		///////////АО КЦ от ШКС-04М////////////////////////////////////////////////////////////////////////
		//{name:АО КЦ от ШКС-04М}
		AOKC_SHKC:singleSignal(table:=ADR(imTable)):=(signal:=di.di_20.bits[0]);
		//{name:Обрыв сигнала "АО КЦ от ШКС-04М"}
		AOKC_SHKC_NS:Reability(table:=ADR(imTable)):=(di1:=di.di_9.bits[3], when:=FALSE);
		//{name:Наличие ЦК "АО КЦ от ШКС-04М"}
		AOKC_SHKC_CK:Reability(table:=ADR(imTable)):=(di1:=di.di_9.bits[3], when:=TRUE);
		
		///////////НО ГПА от кнопки на ШУ////////////////////////////////////////////////////////////////////////
		//{name:НО ГПА от кнопки на ШУ}
		NO_fromSHU:singleSignal(table:=ADR(imTable)):=(signal:=di.di_21.bits[1]);
		//{name:Обрыв сигнала "НО ГПА от кнопки на ШУ"}
		NO_fromSHU_NS:Reability(table:=ADR(imTable)):=(di1:=di.di_9.bits[4], when:=FALSE);
		//{name:Наличие ЦК  "НО ГПА от кнопки на ШУ"}
		NO_fromSHU_CK:Reability(table:=ADR(imTable)):=(di1:=di.di_9.bits[4], when:=TRUE);
		
		///////////АО ГПА от кнопки на ШУ////////////////////////////////////////////////////////////////////////
		//{name:АО ГПА от кнопки на ШУ}
		AO_fromSHU:singleSignal(table:=ADR(imTable)):=(signal:=di.di_21.bits[2]);
		//{name:Обрыв сигнала "АО ГПА от кнопки на ШУ"}
		AO_fromSHU_NS:Reability(table:=ADR(imTable)):=(di1:=di.di_9.bits[5], when:=FALSE);
		//{name:Наличие ЦК  "АО ГПА от кнопки на ШУ"}
		AO_fromSHU_CK:Reability(table:=ADR(imTable)):=(di1:=di.di_9.bits[5], when:=TRUE);
		
		///////////АО ЭГПА от ПРУ////////////////////////////////////////////////////////////////////////
		//{name:АО ЭГПА от ПРУ}
		AO_PRU:singleSignal(table:=ADR(imTable)):=(signal:=di.di_21.bits[3]);
		//{name:Обрыв сигнала "АО ЭГПА от ПРУ"}
		AO_PRU_NS:Reability(table:=ADR(imTable)):=(di1:=di.di_9.bits[6], when:=FALSE);
		//{name:Наличие ЦК "АО ЭГПА от ПРУ"}
		AO_PRU_CK:Reability(table:=ADR(imTable)):=(di1:=di.di_9.bits[6], when:=TRUE);
		
		///////////НКУ ввод 1 включен////////////////////////////////////////////////////////////////////////
		//{name:НКУ ввод 1 включен}
		NKU_1_On:singleSignal(table:=ADR(imTable)):=(signal:=di.di_10.bits[4]);
		//{name:Обрыв сигнала "НКУ ввод 1 включен"}
		NKU_1_On_NS:Reability(table:=ADR(imTable)):=(di1:=di.di_10.bits[4], when:=FALSE);
		//{name:Наличие ЦК  "НКУ ввод 1 включен"}
		NKU_1_On_CK:Reability(table:=ADR(imTable)):=(di1:=di.di_10.bits[4], when:=TRUE);
		
		///////////НКУ ввод 2 включен////////////////////////////////////////////////////////////////////////
		//{name:НКУ ввод 2 включен}
		NKU_2_On:singleSignal(table:=ADR(imTable)):=(signal:=di.di_10.bits[5]);
		//{name:Обрыв сигнала "НКУ ввод 2 включен"}
		NKU_2_On_NS:Reability(table:=ADR(imTable)):=(di1:=di.di_10.bits[5], when:=FALSE);
		//{name:Наличие ЦК  "НКУ ввод 2 включен"}
		NKU_2_On_CK:Reability(table:=ADR(imTable)):=(di1:=di.di_10.bits[5], when:=TRUE);
		///////////Неисправность цепей контроля ИМ////////////////////////////////////////////////////////////////////////
		MVvkl_Obryv_CK_NS:Reability(table:=ADR(imTable)):=(di1:=di.di_7.bits[0], when:=FALSE);
		MVvykl_Obryv_CK_NS:Reability(table:=ADR(imTable)):=(di1:=di.di_7.bits[1], when:=FALSE);
		MVControl_Work_Obryv_CK_NS:Reability(table:=ADR(imTable)):=(di1:=di.di_7.bits[2], when:=FALSE);
		PNS_vkl_CK_NS:Reability(table:=ADR(imTable)):=(di1:=di.di_5.bits[0], when:=FALSE);
		NU1_vkl_CK_NS:Reability(table:=ADR(imTable)):=(di1:=di.di_5.bits[1], when:=FALSE);
		NU2_vkl_CK_NS:Reability(table:=ADR(imTable)):=(di1:=di.di_5.bits[2], when:=FALSE);
		AVOM1_vkl_CK_NS:Reability(table:=ADR(imTable)):=(di1:=di.di_5.bits[3], when:=FALSE);
		AVOM2_vkl_CK_NS:Reability(table:=ADR(imTable)):=(di1:=di.di_5.bits[4], when:=FALSE);
		AVOM3_vkl_CK_NS:Reability(table:=ADR(imTable)):=(di1:=di.di_5.bits[5], when:=FALSE);
		AVOM4_vkl_CK_NS:Reability(table:=ADR(imTable)):=(di1:=di.di_5.bits[6], when:=FALSE);
		TEN_MB_vkl_CK_NS:Reability(table:=ADR(imTable)):=(di1:=di.di_10.bits[0], when:=FALSE);
		TEN_Kollectora_vkl_CK_NS:Reability(table:=ADR(imTable)):=(di1:=di.di_10.bits[1], when:=FALSE);
		Kalorifer_AVOM_vkl_CK_NS:Reability(table:=ADR(imTable)):=(di1:=di.di_10.bits[2], when:=FALSE);
		CMN_vkl_CK_NS:Reability(table:=ADR(imTable)):=(di1:=di.di_10.bits[3], when:=FALSE);
		///////////Наличие цепей контроля ИМ////////////////////////////////////////////////////////////////////////
		MVvkl_NAlichie_CK:Reability(table:=ADR(imTable)):=(di1:=di.di_7.bits[0], when:=TRUE);
		MVvykl_NAlichie_CK:Reability(table:=ADR(imTable)):=(di1:=di.di_7.bits[1], when:=TRUE);
		MVControl_Work_NAlichie_CK:Reability(table:=ADR(imTable)):=(di1:=di.di_7.bits[2], when:=TRUE);
		PNS_vkl_NAlichie_CK:Reability(table:=ADR(imTable)):=(di1:=di.di_5.bits[0], when:=TRUE);
		NU1_vkl_NAlichie_CK:Reability(table:=ADR(imTable)):=(di1:=di.di_5.bits[1], when:=TRUE);
		NU2_vkl_NAlichie_CK:Reability(table:=ADR(imTable)):=(di1:=di.di_5.bits[2], when:=TRUE);
		AVOM1_vkl_NAlichie_CK:Reability(table:=ADR(imTable)):=(di1:=di.di_5.bits[3], when:=TRUE);
		AVOM2_vkl_NAlichie_CK:Reability(table:=ADR(imTable)):=(di1:=di.di_5.bits[4], when:=TRUE);
		AVOM3_vkl_NAlichie_CK:Reability(table:=ADR(imTable)):=(di1:=di.di_5.bits[5], when:=TRUE);
		AVOM4_vkl_NAlichie_CK:Reability(table:=ADR(imTable)):=(di1:=di.di_5.bits[6], when:=TRUE);
		TEN_MB_vkl_NAlichie_CK:Reability(table:=ADR(imTable)):=(di1:=di.di_10.bits[0], when:=TRUE);
		TEN_Kollectora_vkl_NAlichie_CK:Reability(table:=ADR(imTable)):=(di1:=di.di_10.bits[1], when:=TRUE);
		Kalorifer_AVOM_vkl_NAlichie_CK:Reability(table:=ADR(imTable)):=(di1:=di.di_10.bits[2], when:=TRUE);
		CMN_vkl_NAlichie_CK:Reability(table:=ADR(imTable)):=(di1:=di.di_10.bits[3], when:=TRUE);
		///////////Наличие питания////////////////////////////////////////////////////////////////////////
		//{name:Наличие БП1}
		NalichieBP1:singleSignal(table:=ADR(imTable)):=(signal:=di.di_11.bits[0]);
		//{name:Наличие БП2}
		NalichieBP2:singleSignal(table:=ADR(imTable)):=(signal:=di.di_11.bits[1]);
		//{name:Наличие БП3}
		NalichieBP3:singleSignal(table:=ADR(imTable)):=(signal:=di.di_11.bits[2]);
		//{name:Наличие БП4}
		NalichieBP4:singleSignal(table:=ADR(imTable)):=(signal:=di.di_11.bits[3]);
		//{name:Наличие БП5}
		NalichieBP5:singleSignal(table:=ADR(imTable)):=(signal:=di.di_11.bits[4]);
		//{name:Наличие БП6}
		NalichieBP6:singleSignal(table:=ADR(imTable)):=(signal:=di.di_11.bits[5]);
		//{name:Наличие БП7 и БП8}
		NalichieBP7_BP8:singleSignal(table:=ADR(imTable)):=(signal:=di.di_11.bits[6]);
		//{name:Наличие БП9 и БП10}
		NalichieBP9_BP10:singleSignal(table:=ADR(imTable)):=(signal:=di.di_11.bits[7]);
		//{name:Наличие Цепи управления МВ}
		Nalichie_CU_MV:singleSignal(table:=ADR(imTable)):=(signal:=di.di_12.bits[0]);
		//{name:Наличие напряжения  =220 в БРЭО}
		Nalichie220BEAO:singleSignal(table:=ADR(imTable)):=(signal:=di.di_12.bits[1]);
		//{name:Наличие напряжения на входе в ШУ ~220}
		NalichiePer220naVhode:singleSignal(table:=ADR(imTable)):=(signal:=di.di_12.bits[2]);
		//{name:Наличие напряжения на входе в ШУ =220}
		NalichiePost220naVhode:singleSignal(table:=ADR(imTable)):=(signal:=di.di_12.bits[3]);
		//{name:Наличие БП11}
		NalichieBP11:singleSignal(table:=ADR(imTable)):=(signal:=di.di_12.bits[4]);
		//{name:Наличие БП12}
		NalichieBP12:singleSignal(table:=ADR(imTable)):=(signal:=di.di_12.bits[5]);
		
		///////////Отсутствие питания////////////////////////////////////////////////////////////////////////
		//{name:Нет БП1}
		NalichieBP1_NS:singleSignal(table:=ADR(imTable)):=(signal:=di.di_11.bits[0].inverse);
		//{name:Нет БП2}
		NalichieBP2_NS:singleSignal(table:=ADR(imTable)):=(signal:=di.di_11.bits[1].inverse);
		//{name:Нет БП3}
		NalichieBP3_NS:singleSignal(table:=ADR(imTable)):=(signal:=di.di_11.bits[2].inverse);
		//{name:Нет БП4}
		NalichieBP4_NS:singleSignal(table:=ADR(imTable)):=(signal:=di.di_11.bits[3].inverse);
		//{name:Нет БП5}
		NalichieBP5_NS:singleSignal(table:=ADR(imTable)):=(signal:=di.di_11.bits[4].inverse);
		//{name:Нет БП6}
		NalichieBP6_NS:singleSignal(table:=ADR(imTable)):=(signal:=di.di_11.bits[5].inverse);
		//{name:Нет БП7 и БП8}
		NalichieBP7_BP8_NS:singleSignal(table:=ADR(imTable)):=(signal:=di.di_11.bits[6].inverse);
		//{name:Нет БП9 и БП10}
		NalichieBP9_BP10_NS:singleSignal(table:=ADR(imTable)):=(signal:=di.di_11.bits[7].inverse);
		//{name:Нет Цепи управления МВ}
		Nalichie_CU_MV_NS:singleSignal(table:=ADR(imTable)):=(signal:=di.di_12.bits[0].inverse);
		//{name:Нет напряжения  =220 в БРЭО}
		Nalichie220BEAO_NS:singleSignal(table:=ADR(imTable)):=(signal:=di.di_12.bits[1].inverse);
		//{name:Нет напряжения на входе в ШУ ~220}
		NalichiePer220naVhode_NS:singleSignal(table:=ADR(imTable)):=(signal:=di.di_12.bits[2].inverse);
		//{name:Нет напряжения на входе в ШУ =220}
		NalichiePost220naVhode_NS:singleSignal(table:=ADR(imTable)):=(signal:=di.di_12.bits[3].inverse);
		//{name:Нет БП11}
		NalichieBP11_NS:singleSignal(table:=ADR(imTable)):=(signal:=di.di_12.bits[4].inverse);
		//{name:Нет БП12}
		NalichieBP12_NS:singleSignal(table:=ADR(imTable)):=(signal:=di.di_12.bits[5].inverse);
		
		///////////Двери////////////////////////////////////////////////////////////////////////
		//{name:Дверь ШУ открыта Передняя}
		Door_SHU_Front_Open:singleSignal(table:=ADR(imTable)):=(signal:=di.di_13.bits[0]);
		//{name:Дверь ШУ открыта Задняя}
		Door_SHU_Back_Open:singleSignal(table:=ADR(imTable)):=(signal:=di.di_13.bits[1]);
		//{name:БЭАО сработал}
		
		BEAO_Work:singleSignal(table:=ADR(imTable)):=(signal:=di.di_18.bits[1]);
		
		
		//{name:Сброс БЭАО}
		//BEAO_Reset:singleSignal(table:=ADR(imTable)):=(signal:=di.di_18.bits[1]);
		///////////ЩАВР////////////////////////////////////////////////////////////////////////
		//{name:ЩАВР ввод 1 включен}
		SHAVR_1_On:singleSignal(table:=ADR(imTable)):=(signal:=di.di_13.bits[6]);
		//{name:ЩАВР ввод 2 включен}
		SHAVR_2_On:singleSignal(table:=ADR(imTable)):=(signal:=di.di_13.bits[7]);
		
		///////////Кнопки Экстренного останова////////////////////////////////////////////////////////////////////////
		//{name:ЭО ГПА от кнопки на ШУ}
		EO_fromSHU:singleSignal(table:=ADR(imTable)):=(signal:=di.di_14.bits[0]);
		//{name:ЭО ЭГПА от ПРУ}
		EO_PRU:singleSignal(table:=ADR(imTable)):=(signal:=di.di_14.bits[1]);
		
		///////////Напряжение на ИМ////////////////////////////////////////////////////////////////////////
		//{name:Наличие напряжения в ЦУ ПНС}
		NalichieU_PNS:singleSignal(table:=ADR(imTable)):=(signal:=di.di_14.bits[2]);
		//{name:Наличие напряжения в ЦУ НУ1}
		NalichieU_NU1:singleSignal(table:=ADR(imTable)):=(signal:=di.di_14.bits[3]);
		//{name:Наличие напряжения в ЦУ НУ2}
		NalichieU_NU2:singleSignal(table:=ADR(imTable)):=(signal:=di.di_14.bits[4]);
		//{name:Наличие напряжения в ЦУ ЦМН}
		NalichieU_CMN:singleSignal(table:=ADR(imTable)):=(signal:=di.di_14.bits[5]);
		
		///////////Нет Напряжения на ИМ////////////////////////////////////////////////////////////////////////
		//{name:Нет напряжения в ЦУ ПНС}
		NET_U_PNS:singleSignal(table:=ADR(imTable)):=(signal:=di.di_10.bits[10].inverse);
		//{name:Нет напряжения в ЦУ НУ1}
		NET_U_NU1:singleSignal(table:=ADR(imTable)):=(signal:=di.di_10.bits[11].inverse);
		//{name:Нет напряжения в ЦУ НУ2}
		NET_U_NU2:singleSignal(table:=ADR(imTable)):=(signal:=di.di_10.bits[12].inverse);
		//{name:Нет напряжения в ЦУ ЦМН}
		NET_U_CMN:singleSignal(table:=ADR(imTable)):=(signal:=di.di_10.bits[13].inverse);
		
		///////////ИМ в Автомате////////////////////////////////////////////////////////////////////////
		//{name:АВОМ1 в автоматическом режиме}
		AVOM1_Automat:singleSignal(table:=ADR(imTable)):=(signal:=di.di_2.bits[0]);
		//{name:АВОМ2 в автоматическом режиме}
		AVOM2_Automat:singleSignal(table:=ADR(imTable)):=(signal:=di.di_2.bits[1]);
		//{name:АВОМ3 в автоматическом режиме}
		AVOM3_Automat:singleSignal(table:=ADR(imTable)):=(signal:=di.di_2.bits[2]);
		//{name:АВОМ4 в автоматическом режиме}
		AVOM4_Automat:singleSignal(table:=ADR(imTable)):=(signal:=di.di_2.bits[3]);
		
		//{name:ПНС в автоматическом режиме}
		PNS_Automat:singleSignal(table:=ADR(imTable)):=(signal:=di.di_2.bits[4]);
		
		//{name:НУ1 в автоматическом режиме}
		NU1_Automat:singleSignal(table:=ADR(imTable)):=(signal:=di.di_2.bits[5]);
		//{name:НУ2 в автоматическом режиме}
		NU2_Automat:singleSignal(table:=ADR(imTable)):=(signal:=di.di_2.bits[6]);
		
		//{name:ТЭН МБ в автоматическом режиме}
		TEN_MB_Automat:singleSignal(table:=ADR(imTable)):=(signal:=di.di_2.bits[7]);
		//{name:ТЭН Коллектора в автоматическом режиме}
		TEN_Kollectora_Automat:singleSignal(table:=ADR(imTable)):=(signal:=di.di_3.bits[0]);
		
		//{name:Калорифер АВОМ в автоматическом режиме}
		KalAVOM_Automat:singleSignal(table:=ADR(imTable)):=(signal:=di.di_3.bits[1]);
		//{name:ЦМН в автоматическом режиме}
		CMN_Automat:singleSignal(table:=ADR(imTable)):=(signal:=di.di_3.bits[2]);
		//{name:СИнхронизация режима К1}
		Synch_rej_K1:singleSignal(table:=ADR(imTable)):=(signal:=di.di_3.bits[4]);
		Synch_rej_K1_Meandr:singleOutput(table:=ADR(imTable)):=(signal:=od.do_3.bits[13]);
		///////////Поток масла после АВОМ////////////////////////////////////////////////////////////////////////
		//{name:Поток масла после АВОМ > 85 л/мин}
		Flow_Ms_PosleAVOM:singleSignal(table:=ADR(imTable)):=(signal:=di.di_18.bits[0].inverse);
		
		/////////***ДИСКРЕТЫ OUTPUT***//////////////////////////////////////////////////////////////////
		///////////////////////////////////////////////////////////////////////////////////
		
	//	Stop_MV_NO:SingleOutput(table:=ADR(imTable)):=(signal:=od.do_4.bits[2], wait_time:=T#4S);
	
		//{name:Работа ЭГПА}
		Work_EGPA:SingleOutput(table:=ADR(imTable)):=(signal:=od.do_4.bits[2]);
		//{name:Неисправность ЭГПА}
		Neispr_EGPA:SingleOutput(table:=ADR(imTable)):=(signal:=od.do_4.bits[0]);
		//{name:Авария ЭГПА}
		Avary_EGPA:SingleOutput(table:=ADR(imTable)):=(signal:=od.do_4.bits[1]);
		//{name:Наличие напряжения лампа на двери}
		U_Lamp_SHU:SingleOutput(table:=ADR(imTable)):=(signal:=od.do_4.bits[3]);
			//{name:Посветка кнопки при АО}
		AO_Knopka_ind:SingleOutput(table:=ADR(imTable)):=(signal:=od.do_4.bits[4]);
		//{name:Пуск в ШУП}
		Pusk_SHUP:SingleOutput(table:=ADR(imTable)):=(signal:=od.do_4.bits[8], wait_time:=T#4S);
		//{name:Останов в ШУП}
		Stop_SHUP:SingleOutput(table:=ADR(imTable)):=(signal:=od.do_4.bits[9], wait_time:=T#4S);
		//{name:Фонарь НО}
		NO_Fonar:SingleOutput(table:=ADR(imTable)):=(signal:=od.do_3.bits[10]);
		//{name:Фонарь ПС}
		PC_Fonar:SingleOutput(table:=ADR(imTable)):=(signal:=od.do_3.bits[9]);
		//{name:Фонарь АС}
		AC_Fonar:SingleOutput(table:=ADR(imTable)):=(signal:=od.do_3.bits[8]);
		//{name:смазка крана 1}
		Kr1_Smazka:SingleOutput(table:=ADR(imTable)):=(signal:=od.do_0.bits[14], wait_time:=T#15S);
		//{name:смазка крана 2}
		Kr2_Smazka:SingleOutput(table:=ADR(imTable)):=(signal:=od.do_0.bits[15], wait_time:=T#15S);
		//{name:Кран 4 открыть из 3 этапа пуска}
		Kr_4_Open_From_Alg:SingleOutput(table:=ADR(imTable)):=(signal:=od.do_0.bits[8]);
		/////////***ДИСКРЕТЫ Неисправности***//////////////////////////////////////////////////////////////////
	
		
		
		/////////***НАличие Цепей контроля***//////////////////////////////////////////////////////////////////
		///////////////////////////////////////////////////////////////////////////////////
		
		
	END_STRUCT
END_TYPE

// K1/std12k5/hardwareConfig/DiConfig
TYPE DiConfig:
	STRUCT
		di_0:DiSourceMlp(table:=ADR(kontroller.inputTable)):=(addr:=0);//
		di_1:DiSourceMlp(table:=ADR(kontroller.inputTable)):=(addr:=1);//
		di_2:DiSourceMlp(table:=ADR(kontroller.inputTable)):=(addr:=2);//
		di_3:DiSourceMlp(table:=ADR(kontroller.inputTable)):=(addr:=3);//
		di_4:DiSourceMlp(table:=ADR(kontroller.inputTable)):=(addr:=4);//
		di_5:DiSourceMlp(table:=ADR(kontroller.inputTable)):=(addr:=5);//
		di_6:DiSourceMlp(table:=ADR(kontroller.inputTable)):=(addr:=6);//
		di_7:DiSourceMlp(table:=ADR(kontroller.inputTable)):=(addr:=7);//
		di_8:DiSourceMlp(table:=ADR(kontroller.inputTable)):=(addr:=8);//
		di_9:DiSourceMlp(table:=ADR(kontroller.inputTable)):=(addr:=9);//
		di_10:DiSourceMlp(table:=ADR(kontroller.inputTable)):=(addr:=10);//
		di_11:DiSourceMlp(table:=ADR(kontroller.inputTable)):=(addr:=11);//
		di_12:DiSourceMlp(table:=ADR(kontroller.inputTable)):=(addr:=12);//
		di_13:DiSourceMlp(table:=ADR(kontroller.inputTable)):=(addr:=13);//
		di_14:DiSourceMlp(table:=ADR(kontroller.inputTable)):=(addr:=14);//
		di_15:DiSourceMlp(table:=ADR(kontroller.inputTable)):=(addr:=15);//
		di_16:DiSourceMlp(table:=ADR(kontroller.inputTable)):=(addr:=16);//
		di_17:DiSourceMlp(table:=ADR(kontroller.inputTable)):=(addr:=17);//
		di_18:DiSourceMlp(table:=ADR(kontroller.inputTable)):=(addr:=18);//
		di_19:DiSourceMlp(table:=ADR(kontroller.inputTable)):=(addr:=19);//
		di_20:DiSourceMlp(table:=ADR(kontroller.inputTable)):=(addr:=20);//
		di_21:DiSourceMlp(table:=ADR(kontroller.inputTable)):=(addr:=21);//
	
	END_STRUCT
END_TYPE

// K1/std12k5/modbus/MbsConfig
TYPE MbsConfig:
	STRUCT
		devName:tstModbus(table:=ADR(kontrollers)):=(mbRole:=MbKontrollerRole.MK_SLAVE);

	END_STRUCT
END_TYPE

// lowLevel_ecl/Common/parameters/question/Answers
TYPE Answers :
(
	ANS_NONE	:=	16#00,
	ANS_YES		:=	16#01,
	ANS_NO		:=	16#02,
	ANS_CANCEL	:=	16#04,
	ANS_RETRY	:=	16#08
) UINT;
END_TYPE

// lowLevel_ecl/kontroller/baseSources/statusAi
TYPE statusAi :
(
	NOTDEFINED:=0,
	LL:=1,
	HL:=2,
	NOTRELIABLE:=3,
	normal:=4,
	LW:=5,
	HW:=6,
	LA:=7,
	HA:=8
		
) BYTE;
END_TYPE

// lowLevel_ecl/kontroller/extSources/MultiAnalogLimits
TYPE MultiAnalogLimits :
(
	SELF := 0,
	ANY_INPUT:=1,
	ALL_INPUTS:=2
);
END_TYPE

// lowLevel_ecl/kontroller/mlp/sDIN_DOUT
TYPE sDIN_DOUT :
STRUCT

	s_Aux	:	WORD	;	//	bit-0 присутствие 1-есть, 0 -нет (привязка в конфигурации MLP)
							//	bit-1 тип модуля 1-выходной, 0 -входной
							//	bit-2 достоверность 1- достоверно,0- не достоверно
									  
	kcc		:	WORD	;   //	Контроль Целостности Цепи - КЦЦ
							//	каждая цепь 2 бита
							//	00 - неизвестно или обрыв цепи
							//	01 - есть Целостность Цепи
							//	10 - есть ток
							//	11 - КЗ
									  
	kk		:	WORD	;	//	Контроль выхода команды - КК
							//	каждая цепь 2 бита
							//	00 - не бывает
							//	01 - пассивное состояние
							//	10 - активное (есть выход)состояние
							//	11 - ошибка выхода команды 
									  
	value_cc:	WORD	;	//	содержимое выходных регистров 

END_STRUCT
END_TYPE

// lowLevel_ecl/kontroller/mlp/AIn_s
TYPE AIn_s :
STRUCT
	
f	:	DWORD	;	//	bit-0 присутствие в проекте MLP. 1-есть, 0 –нет
					//	bit-1 тип модуля 1-выходной, 0 -входной
					//	bit-2 достоверность 1- достоверно,0- не достоверно. Диагностика общая: и по диапазонам измерения, и собственная по каналу модуля.
					//	bit-3 размерность сигнала 1- в физических величинах,0- значение тока (0-20100)
					//	bit-4 1- ниже нижней границы,0 - выше нижней границы
					//	bit-5 1- выше верхней границы,0 - ниже верхней границы
					//	bit-6 1- общий бит отказа канала( по ИЛИ Not(bit2), bit4, bit5)

val	:	REAL	;	//	Значение аналогового входа 4-20мА - 40000-20000 


END_STRUCT
END_TYPE

// lowLevel_ecl/kontroller/mlp/DIn_s
TYPE DIn_s :
STRUCT
	
f	:	WORD	;	//	bit-0 присутствие в проекте MLP. 1-есть, 0 -нет
					//	bit-1 тип модуля 1-выходной, 0 -входной
					//	bit-2 достоверность 1- достоверно,0- не достоверно 

val	:	WORD	;	//	Контроль канала
					//	Каждая цепь 2 бита
	                //	00 - обыв цепи
					//	01 - недостоверно
					//	10 - контакт разомкнут
					//	11 - контакт замкнут	

END_STRUCT
END_TYPE

// lowLevel_ecl/kontroller/mlp/sAIN_AOUT
TYPE sAIN_AOUT :
STRUCT

s_Aux	:	WORD	;	//	bit-0 присутствие 1-есть, 0 -нет
						//	bit-1 тип модуля 1-выходной, 0 -входной
						//	bit-2 достоверность 1- достоверно,0- не достоверно
						//	bit-3 0- значение тока (0-20100)
						
s_value	:	REAL	;	//	Действительный (измеренный) выходной ток 4-20мА - 4000-20000

END_STRUCT
END_TYPE

// lowLevel_ecl/kontroller/mlp/TypeUSO
TYPE TypeUSO :
(
	NotUso, DIN, DOUT, AIN, AOUT, RS485
);
END_TYPE

// lowLevel_ecl/kontroller/mlp/DiagnosticIndex
TYPE DiagnosticIndex :
STRUCT
	Index: INT; // Индекс первого канала в MLP модуля УСО
	TypeModule: TypeUSO; // Тип модуля УСО
	FirstNomComPort: WORD; // Первый номер COM порта модуля RS485 
END_STRUCT
END_TYPE

// lowLevel_ecl/kontroller/mlp/Diagnostic/iniFile/iniFileLine
TYPE iniFileLine :
STRUCT
	status:iniFileStatus;
	Section:STRING;
	Parameter:STRING;
	Value:STRING;
END_STRUCT
END_TYPE

// lowLevel_ecl/kontroller/mlp/Diagnostic/iniFile/iniFileStatus
TYPE iniFileStatus :
(
	NotDefined,
	Section,
	Parametr,
	Eof
);
END_TYPE

// lowLevel_ecl/kontroller/mlp/Diagnostic/BsDescriptor
TYPE BsDescriptor :
STRUCT
	enabled:bool;
//	modules:ARRAY[1..15] OF ModuleDescriptor;
	modules:ARRAY[1..16] OF ModuleDescriptor;
END_STRUCT
END_TYPE

// lowLevel_ecl/kontroller/mlp/Diagnostic/ModuleDescriptor
TYPE ModuleDescriptor :
STRUCT
	moduleType:ModuleTypes;
	addr:WORD;
	addrB:WORD;
	funct:BYTE;
END_STRUCT
END_TYPE

// lowLevel_ecl/kontroller/mlp/Diagnostic/BsStatusDecriptor
TYPE BsStatusDecriptor :
STRUCT
	connected:BOOL;
//	modules:ARRAY[1..15] OF ModuleStatusDescriptor;
	modules:ARRAY[1..16] OF ModuleStatusDescriptor;
END_STRUCT
END_TYPE

// lowLevel_ecl/kontroller/mlp/Diagnostic/ModuleStatusDescriptor
TYPE ModuleStatusDescriptor :
STRUCT
	moduleStatus:WORD;
	pinStatus: WORD;
END_STRUCT
END_TYPE

// lowLevel_ecl/kontroller/mlp/Diagnostic/ModuleTypes
TYPE ModuleTypes :
(
	    none:=0,
        DI8:=16#4002,
        DO5:=16#1502,
        AI4:=16#2002,
		OA4:=16#3002,
		RS485:=16#0020,
		IF3:=16#1903
) WORD;
END_TYPE

// lowLevel_ecl/kontroller/baseSources/AnalogAlarms
TYPE AnalogAlarms :
(
	NONE:=0,
	LW:=16#1,
	HW:=16#2,
	LA:=16#4,
	HA:=16#8,
	ALL:=16#F
) BYTE;
END_TYPE

// lowLevel_ecl/kontroller/baseSources/AnalogLimitFlags
TYPE AnalogLimitFlags :
(
	NONE:=0,
	LL:=16#1,
	LW:=16#2,
	HW:=16#4,
	LA:=16#8,
	HA:=16#10,
	HL:=16#20
) BYTE;
END_TYPE

// lowLevel_ecl/im/BaseIms/cmdSources
TYPE cmdSources : 
(
	Algoritm := 0,
	ARM:=1,
	MPU:=2,
	LPU:=3
) UINT;
END_TYPE

// lowLevel_ecl/im/BaseIms/statusDualInput
TYPE statusDualInput :
(
	STATUS_NOTDEFINED:=0,
	STATUS_ON:=1,
	STATUS_OFF:=2,
	STATUS_TRANSITIONAL:=3,
	STATUS_ERROR:=4
) BYTE;
END_TYPE

// REZERV1/RezervState
TYPE RezervState :
( Nothing:=0, Single:=1, Active:=2, Passive:=3
//	enum_member := 4
) WORD;
END_TYPE

// K1/std12k5/algoritms/ModeGpa
TYPE ModeGpa :
(
	MODE_NOTDEFINED	:= 0, //РЕЖИМ НЕ определен
	MODE_STOP		:= 1, //ГПА остановлен
	MODE_PUSKAP_R	:= 2, //Автоматический пуск Рекакторный
	MODE_PUSKPP_R	:= 3, //Поэтапный пуск Рекакторный
	MODE_PUSKAP_Ch	:= 4, //Автоматический пуск Рекакторный
	MODE_PUSKPP_Ch	:= 5, //Поэтапный пуск Рекакторный
	MODE_WORK_M		:= 6, //Работа в магистраль
	MODE_WORK_K		:= 7, //Работа в кольцо
	MODE_NO			:= 8, //Режим НО
	MODE_AO			:= 9, //Режим АО
	MODE_EO			:= 10, //Режим ЭО
	MODE_TESTIM		:= 11, //Режим тест ИМ
	MODE_PUSKV_R	:= 12, //Режим проверка двигателя в реакторном режиме
	MODE_PUSKV_Ch	:= 13, //Режим проверка двигателя в частотном режиме
	MODE_PUSKK		:= 14, //Режим проверка кранов
	MODE_PROVPMS	:= 15, //Режим проверка давления маслосмазки
	MODE_PROBDPMG	:= 16,	//Режим проверка перепад масло-газ
	MODE_I			:= 17, //режим имитации пуска
	MODE_O			:= 18, //режим опрессовки
	TEST_PROTECTIONS:= 19 //Режим тест защит
) UINT;
END_TYPE

// K1/std12k5/algoritms/ProtectionsConfig
TYPE ProtectionsConfig:
		{attribute 'symbol' := 'read'}
	STRUCT
	(*Температуры т.1 - т.10*) 
		p_TOpornogoPodshipnikaEDT_1:AiProtection (table:=protectManager.getTable())							:=(ai:=ai.TOpornogoPodshipnikaEDT_1	,controlLimit:=statusAi.HA,delay:=(value:=T#3S));
		p_TOpornoYpornogoPodshipnikaEDT_2:AiProtection (table:=protectManager.getTable())					:=(ai:=ai.TOpornoYpornogoPodshipnikaEDT_2 ,controlLimit:=statusAi.HA,delay:=(value:=T#3S));
		p_TOpornoYpornogoPodshipnikaKolesaRedEDT_3:AiProtection (table:=protectManager.getTable())			:=(ai:=ai.TOpornoYpornogoPodshipnikaKolesaRedEDT_3,controlLimit:=statusAi.HA,delay:=(value:=T#3S));
		p_TOpornoYpornogoPodshipnikaKolesaRedHT_4:AiProtection (table:=protectManager.getTable())			:=(ai:=ai.TOpornoYpornogoPodshipnikaKolesaRedHT_4,controlLimit:=statusAi.HA,delay:=(value:=T#3S));
		p_TOpornogoPodshipnikaShesterniReduktoraT_5:AiProtection (table:=protectManager.getTable())			:=(ai:=ai.TOpornogoPodshipnikaShesterniReduktoraT_5	,controlLimit:=statusAi.HA,delay:=(value:=T#3S));
		p_TOpornogoPodshipnikaReduktoraHT_6:AiProtection (table:=protectManager.getTable())					:=(ai:=ai.TOpornogoPodshipnikaReduktoraHT_6,controlLimit:=statusAi.HA,delay:=(value:=T#3S));
		p_TOpornoYpornogoPodshipnikaNagnetateljaT_7:AiProtectionDual (table:=protectManager.getTable())		:=(	ai1:=ai.TOpornoYpornogoPodshipnikaNagnetateljaT_7_1,
																											ai2:=ai.TOpornoYpornogoPodshipnikaNagnetateljaT_7_2	,
																											controlLimit:=statusAi.HA, 
																											control_Normal:=statusAi.Normal, 
																											delay:=(value:=T#3S));
		p_TOpornoYpornogoPodshipnikaSvobodnogoKoncaNT_8:AiProtectionDual (table:=protectManager.getTable())	:=(	ai1:=ai.TOpornoYpornogoPodshipnikaSvobodnogoKoncaNT_8_1,
																											ai2:=ai.TOpornoYpornogoPodshipnikaSvobodnogoKoncaNT_8_2	,
																											controlLimit:=statusAi.HA, 
																											control_Normal:=statusAi.Normal, 
																											delay:=(value:=T#3S));
		p_TYpornogoPodshipnikaRavKolodokHT_9:AiProtectionDual (table:=protectManager.getTable())				:=(	ai1:=ai.TYpornogoPodshipnikaRavKolodokHT_9_1,
																											ai2:=ai.TYpornogoPodshipnikaRavKolodokHT_9_2,
																											controlLimit:=statusAi.HA, 
																											control_Normal:=statusAi.Normal, 
																											delay:=(value:=T#3S));
		p_TYpornogoPodshipnikaNerabKolodokHT_10:AiProtectionDual (table:=protectManager.getTable())				:=(	ai1:=ai.TYpornogoPodshipnikaNerabKolodokHT_10_1,
																											ai2:=ai.TYpornogoPodshipnikaNerabKolodokHT_10_2,
																											controlLimit:=statusAi.HA, 
																											control_Normal:=statusAi.Normal, 
																											delay:=(value:=T#3S));
		p_TgazaNaVyhodeH:AiProtection (table:=protectManager.getTable())									:=(ai:=ai.TgazaNaVyhodeH,controlLimit:=statusAi.HA,delay:=(value:=T#3S));
		
	(*Давления*)
		
		p_OsSdvigNagnetatelja_Plus:AiProtection (table:=protectManager.getTable())							:=(ai:=ai.OsSdvigNagnetatelja_Plus,controlLimit:=statusAi.HA,delay:=(value:=T#3S));
		p_OsSdvigNagnetatelja_Minus:AiProtection (table:=protectManager.getTable())							:=(ai:=ai.OsSdvigNagnetatelja_Minus,controlLimit:=statusAi.HA,delay:=(value:=T#3S));
		p_DGazaNaVhodeNagnetatelja_GPA_STOP:AiProtection (table:=protectManager.getTable())					:=(ai:=ai.DGazaNaVhodeNagnetatelja,controlLimit:=statusAi.normal,ControlValue:=0.3, delay:=(value:=T#3S));
		p_DGazaNaVyhodeNagnetatelja_GPA_STOP:AiProtection (table:=protectManager.getTable())				:=(ai:=ai.DGazaNaVyhodeNagnetatelja,controlLimit:=statusAi.normal,ControlValue:=0.3, delay:=(value:=T#3S));
		//p_DGazaNaVhodeNagnetatelja:AiProtection (table:=protectManager.getTable())							:=(ai:=ai.DGazaNaVhodeNagnetatelja,controlLimit:=statusAi.LA,delay:=(value:=T#3S));
		p_DGazaNaVyhodeNagnetatelja:AiProtection (table:=protectManager.getTable())							:=(ai:=ai.DGazaNaVyhodeNagnetatelja,controlLimit:=statusAi.HA,delay:=(value:=T#3S));
		p_PerepadDavlenieMasloGaz:AiProtection (table:=protectManager.getTable())							:=(ai:=ai.PerepadDavlenieMasloGaz,controlLimit:=statusAi.LA, delay:=(value:=T#20S));
		p_DavlenijaMasloSmNizkoe:AiProtection (table:=protectManager.getTable())							:=(ai:=ai.DavlenijaMasloSmNizkoe,controlLimit:=statusAi.LA, delay:=(value:=T#16S));
		p_DavlenijaMasloSmVysokoe:AiProtection (table:=protectManager.getTable())							:=(ai:=ai.DavlenijaMasloSmVysokoe,controlLimit:=statusAi.LA, delay:=(value:=T#16S));
	
	(*Вибрация*)
		
		p_VibroSkorostOPED_T1:AiProtection (table:=protectManager.getTable())								:=(ai:=ai.VibroSkorostOPED_T1,controlLimit:=statusAi.HA,delay:=(value:=T#3S));
		p_VibroSkorostOYPED_T2:AiProtection (table:=protectManager.getTable())								:=(ai:=ai.VibroSkorostOYPED_T2,controlLimit:=statusAi.HA,delay:=(value:=T#3S));
		p_VibroSkorostOYPKolesaED_T3:AiProtection (table:=protectManager.getTable())						:=(ai:=ai.VibroSkorostOYPKolesaED_T3,controlLimit:=statusAi.HA,delay:=(value:=T#3S));
		p_VibroSkorostOPKolesaRH_T4:AiProtection (table:=protectManager.getTable())							:=(ai:=ai.VibroSkorostOPKolesaRH_T4	,controlLimit:=statusAi.HA,delay:=(value:=T#3S));
		p_VibroSkorostOPShesterniRED_T5:AiProtection (table:=protectManager.getTable())						:=(ai:=ai.VibroSkorostOPShesterniRED_T5	,controlLimit:=statusAi.HA,delay:=(value:=T#3S));
		p_VibroSkorostOPShesterniReduktoraH_T6:AiProtection (table:=protectManager.getTable())				:=(ai:=ai.VibroSkorostOPShesterniReduktoraH_T6,controlLimit:=statusAi.HA,delay:=(value:=T#3S));
	(*Дискретные сигналы *)
		
		p_PerepadDavlenieMasloGaz_Less100:DiProtection (table:=protectManager.getTable())					:=(di:=Im.PerepadDavlenieMasloGaz_Less100,when:=TRUE, delay:=(value:=T#20S));
		p_RegVozbOff:DiProtection (table:=protectManager.getTable())										:=(di:=Im.RegVozbOff, when:=TRUE,delay:=(value:=T#3S));
		p_Fail_Chastotniy_Pusk:DiProtection (table:=protectManager.getTable())								:=(di:=Im.Fail_Chastotniy_Pusk, when:=TRUE,delay:=(value:=T#1S));
		p_OFFAvarSwitch:DiProtection (table:=protectManager.getTable())										:=(di:=Im.OFFAvarSwitch,when:=TRUE,delay:=(value:=T#1S));
		p_AOKC_SHKC:DiProtection (table:=protectManager.getTable())											:=(di:=Im.AOKC_SHKC	,when:=TRUE,delay:=(value:=T#1S));
		p_AO_PRU:DiProtection (table:=protectManager.getTable())											:=(di:=Im.AO_PRU	,when:=TRUE);
		p_AO_fromSHU:DiProtection (table:=protectManager.getTable())										:=(di:=Im.AO_fromSHU	,when:=TRUE);	
					
(*Защиты по ИМ *)																							
		p_mvOff:MvProtection(table:=protectManager.getTable())												:=(sw:=Im.mv,delay:=(value:=T#1S));
		p_kran1:Krans_Protections(table:=protectManager.getTable())											:=(Krans:=Im.kran1, delay:=(value:=T#10S), dP_Konf:=ystavki.dP_Konf_kr1);
		p_kran2:Krans_Protections(table:=protectManager.getTable())											:=(Krans:=Im.kran2, delay:=(value:=T#10S), dP_Konf:=ystavki.dP_Konf_kr1);
		
	END_STRUCT
END_TYPE

// lowLevel_ecl/kontroller/extSources/AnalogItem
TYPE AnalogItem :
STRUCT
	input: REFERENCE TO AISource; 
END_STRUCT
END_TYPE

// K1/std12k5/algoritms/YstavkiConfig
TYPE YstavkiConfig:
		{attribute 'symbol' := 'read'} 
	STRUCT
		blockkr1: (*REFERENCE TO*)  DiscretParametr (table:=ADR(YstTable)) ;//{name:блокировать самосдвиг крана 1}
		blockkr2:(*REFERENCE TO*) DiscretParametr (table:=ADR(YstTable));//{name:блокировать самосдвиг крана 2}
		blockkr3:(*REFERENCE TO*) DiscretParametr (table:=ADR(YstTable));//{name:блокировать самосдвиг крана 3}
		blockkr3b:(*REFERENCE TO*) DiscretParametr (table:=ADR(YstTable));//{name:блокировать самосдвиг крана 3б}
		blockkr4:(*REFERENCE TO*) DiscretParametr (table:=ADR(YstTable));//{name:блокировать самосдвиг крана 4}
		blockkr5:(*REFERENCE TO *)DiscretParametr (table:=ADR(YstTable));//{name:блокировать самосдвиг крана 5}
		blockkr6:(*REFERENCE TO *)DiscretParametr (table:=ADR(YstTable));//{name:блокировать самосдвиг крана 6}
		Block_kr4_alg:DiscretParametr (table:=ADR(YstTable));
		Block_kr1_alg:DiscretParametr (table:=ADR(YstTable));
		Block_kr2_alg:DiscretParametr (table:=ADR(YstTable));
		Block_kr3_alg:DiscretParametr (table:=ADR(YstTable));
		Block_kr3b_alg:DiscretParametr (table:=ADR(YstTable));
		Block_kr5_alg:DiscretParametr (table:=ADR(YstTable));
		Block_kr6_alg:DiscretParametr (table:=ADR(YstTable));
		
		block_OPC_cmd:DiscretParametr (table:=ADR(YstTable));
		
		////////////////////ПС по СИП//////////////////////////////////////////////////////
		SIp_T1: SIP_PS (table:=ADR(YstTable)):=(ai:= ai.TOpornogoPodshipnikaEDT_1);
		
		SIp_T2: SIP_PS (table:=ADR(YstTable)):=(ai:= ai.TOpornoYpornogoPodshipnikaEDT_2);
		
		SIp_T3: SIP_PS (table:=ADR(YstTable)):=(ai:= ai.TOpornoYpornogoPodshipnikaKolesaRedEDT_3);
		
		SIp_T4: SIP_PS (table:=ADR(YstTable)):=(ai:= ai.TOpornoYpornogoPodshipnikaKolesaRedHT_4);
		
		SIp_T5: SIP_PS (table:=ADR(YstTable)):=(ai:= ai.TOpornogoPodshipnikaShesterniReduktoraT_5);
		
		SIp_T6: SIP_PS (table:=ADR(YstTable)):=(ai:= ai.TOpornogoPodshipnikaReduktoraHT_6);
		
		SIp_T7_1: SIP_PS (table:=ADR(YstTable)):=(ai:= ai.TOpornoYpornogoPodshipnikaNagnetateljaT_7_1);
		
		SIp_T7_2: SIP_PS (table:=ADR(YstTable)):=(ai:= ai.TOpornoYpornogoPodshipnikaNagnetateljaT_7_2);
		
		SIp_T8_1: SIP_PS (table:=ADR(YstTable)):=(ai:= ai.TOpornoYpornogoPodshipnikaSvobodnogoKoncaNT_8_1);
		
		SIp_T8_2: SIP_PS (table:=ADR(YstTable)):=(ai:= ai.TOpornoYpornogoPodshipnikaSvobodnogoKoncaNT_8_2);
		
		SIp_T9_1: SIP_PS (table:=ADR(YstTable)):=(ai:= ai.TYpornogoPodshipnikaRavKolodokHT_9_1	);
		
		SIp_T9_2: SIP_PS (table:=ADR(YstTable)):=(ai:= ai.TYpornogoPodshipnikaRavKolodokHT_9_2	);
		
		SIp_T10_1: SIP_PS (table:=ADR(YstTable)):=(ai:= ai.TYpornogoPodshipnikaNerabKolodokHT_10_1	);
		
		SIp_T10_2: SIP_PS (table:=ADR(YstTable)):=(ai:= ai.TYpornogoPodshipnikaNerabKolodokHT_10_2	);
		
		SIp_T_Vyhode_N: SIP_PS (table:=ADR(YstTable)):=(ai:= ai.TgazaNaVyhodeH);
		
		SIp_T_Posle_AVOM: SIP_PS (table:=ADR(YstTable)):=(ai:= ai.TMaslaPosleAVOM);
		
		SIp_T_Masla_MB: SIP_PS (table:=ADR(YstTable)):=(ai:= ai.TMaslaMB);
		
		SIp_T_Masla_TEN: SIP_PS (table:=ADR(YstTable)):=(ai:= ai.TMaslaMB_TEN);
		
		////////////////////НАРАБОТКА//////////////////////////////////////////////////////
		
		nu1_narab: nu1 (table:=ADR(YstTable));		
		nu2_narab: nu2 (table:=ADR(YstTable));
		//pns_narab: pns_ (table:=ADR(YstTable));
		Work_HRS: work (table:=ADR(YstTable));
		Pusk_times: pusk (table:=ADR(YstTable));
		AO_times: AO (table:=ADR(YstTable));
		NO_times: NO (table:=ADR(YstTable));
		EO_times: EO (table:=ADR(YstTable));
		//CMN_Narab:CMN (table:=ADR(YstTable));
		//Kalorifer_AVOM_Narab: Kalorifer_AVOM (table:=ADR(YstTable));
		//TEN_Kollectora_narab: TEN_Kollectora (table:=ADR(YstTable));
	//	TEN_MB_Narab:			TEN_MB (table:=ADR(YstTable));
		////////////////////Уставки//////////////////////////////////////////////////////
		YstPNS_YP:  AutoPNS_YP (table:=ADR(YstTable));
		YstPNS_YT:  AutoPNS_YT (table:=ADR(YstTable));
		
		Yst_Vkl_TEN:	AutoTEN_YP (table:=ADR(YstTable));
		Yst_Vykl_TEN:	AutoTEN_YT (table:=ADR(YstTable));
		
		Yst_AVOM_T1:	T1_AVOM (table:=ADR(YstTable));
		Yst_AVOM_T2:	T2_AVOM (table:=ADR(YstTable));
		Yst_AVOM_T3:	T3_AVOM (table:=ADR(YstTable));
		Yst_AVOM_T4:	T4_AVOM (table:=ADR(YstTable));
		
		Yst_Tvkl_AVOM1:	Tvkl_AVOM1 (table:=ADR(YstTable));
		Yst_Tvkl_AVOM2:	Tvkl_AVOM2 (table:=ADR(YstTable));
		Yst_Tvkl_AVOM3:	Tvkl_AVOM3 (table:=ADR(YstTable));
		Yst_Tvkl_AVOM4:	Tvkl_AVOM4 (table:=ADR(YstTable));
		
		Yst_Tvykl_AVOM1:	Tvykl_AVOM1 (table:=ADR(YstTable));
		Yst_Tvykl_AVOM2:	Tvykl_AVOM2 (table:=ADR(YstTable));
		Yst_Tvykl_AVOM3:	Tvykl_AVOM3 (table:=ADR(YstTable));
		Yst_Tvykl_AVOM4:	Tvykl_AVOM4 (table:=ADR(YstTable));
		
		Yst_DTvykl_AVOM1:	Delta_Vykl_AVOM1 (table:=ADR(YstTable));
		Yst_DTvykl_AVOM2:	Delta_Vykl_AVOM2 (table:=ADR(YstTable));
		Yst_DTvykl_AVOM3:	Delta_Vykl_AVOM3 (table:=ADR(YstTable));
		Yst_DTvykl_AVOM4:	Delta_Vykl_AVOM4 (table:=ADR(YstTable));
		
		num_Avom:			Number_Of_Avom (table:=ADR(YstTable));
		
		////////////////////Управляющие сигналы//////////////////////////////////////////////////////
		//{name:рассогласование аналогов и дискрета по dPм-г}
		dPmg_Rassogl: Rassoglasovanie_dPmg (table:=ADR(YstTable)):=(di:=im.PerepadDavlenieMasloGaz_Less100, ai:=AI.PerepadDavlenieMasloGaz);
		dP_Konf_kr1:DiscretParametr (table:=ADR(YstTable));	
		dP_Konf_kr2:DiscretParametr (table:=ADR(YstTable));	
		(*sip_t1_new:SEt_New_SIP (table:=ADR(YstTable)):=(Ai:=ai.TOpornogoPodshipnikaEDT_1, n:= 0);*)
	END_STRUCT
END_TYPE

// K2/std12k5/hardwareConfig/AOConfig
TYPE AOConfig:
	STRUCT
		//AoName:AoSourceMlp(table:=ADR(kontroller.outputTable)):=(addr:=0);
	END_STRUCT
END_TYPE

// K2/std12k5/hardwareConfig/DOConfig
TYPE DOConfig:
	STRUCT
		do_0:DoSourceMlp(table:=ADR(kontroller.outputTable)):=(addr:=0);
		do_1:DoSourceMlp(table:=ADR(kontroller.outputTable)):=(addr:=1);
		do_2:DoSourceMlp(table:=ADR(kontroller.outputTable)):=(addr:=2);
		do_3:DoSourceMlp(table:=ADR(kontroller.outputTable)):=(addr:=3);
		do_4:DoSourceMlp(table:=ADR(kontroller.outputTable)):=(addr:=4);	
	END_STRUCT
END_TYPE

// K2/std12k5/hardwareConfig/AiConfig
TYPE AiConfig:
	STRUCT
		///////////////////////////////////////////////////////////////////////////////////////////////////////////////
		//{name:Температура стали статора 1 канал}
		TStalisStatoraKanall:AI_Final(table:=ADR(kontroller.inputTable)):=(addr:=0, dLL:=0,dHL:=150, dHW:=130, histeresis:=0.5);
		//{name:Температура стали статора 2 канал}
		TStalisStatoraKanal2:AI_Final(table:=ADR(kontroller.inputTable)):=(addr:=1, dLL:=0,dHL:=150, dHW:=130, histeresis:=0.5);
		//{name:Температура стали статора 3 канал}
		TStalisStatoraKanal3:AI_Final(table:=ADR(kontroller.inputTable)):=(addr:=2, dLL:=0,dHL:=150, dHW:=130, histeresis:=0.5);
	
		///////////////////////////////////////////////////////////////////////////////////////////////////////////////
		//{name:Температура меди статора 1 канал}
		TMediStatoraKanall:AI_Final(table:=ADR(kontroller.inputTable)):=(addr:=3, dLL:=0,dHL:=150, dHW:=130, histeresis:=0.5);
		//{name:Температура меди статора 2 канал}
		TMediStatoraKanal2:AI_Final(table:=ADR(kontroller.inputTable)):=(addr:=4, dLL:=0,dHL:=150, dHW:=130, histeresis:=0.5);
		//{name:Температура меди статора 3 канал}
		TMediStatoraKanal3:AI_Final(table:=ADR(kontroller.inputTable)):=(addr:=5, dLL:=0,dHL:=150, dHW:=130, histeresis:=0.5);
		
		
	
		
		///////////////////////////////////////////////////////////////////////////////////////////////////////////////
		//{name:Температура опорного подшипника ЭД т.1 }
		TOpornogoPodshipnikaEDT_1:AI_Final_SIP(table:=ADR(kontroller.inputTable)):=(addr:=6, dLL:=0,dHL:=100,dHW:=75,dHA:=80,  histeresis:=0.5, ChangeSIP:=(value:=10));
		//{name:Температура опорно-упорного подшипника ЭД т.2}
		TOpornoYpornogoPodshipnikaEDT_2:AI_Final_SIP(table:=ADR(kontroller.inputTable)):=(addr:=7,dLL:=0,dHL:=100,dHW:=75,dHA:=80, histeresis:=0.5, ChangeSIP:=(value:=10));
		//{name:Температура опорно-упорного подшипника колеса редуктора со стороны ЭД т.3}
		TOpornoYpornogoPodshipnikaKolesaRedEDT_3:AI_Final_SIP(table:=ADR(kontroller.inputTable)):=(addr:=8, dLL:=0,dHL:=100,dHW:=75,dHA:=80,  histeresis:=0.5, ChangeSIP:=(value:=10));
		//{name:Температура опорно-упорного подшипника колеса редуктора со стороны Нагнетателя т.4}
		TOpornoYpornogoPodshipnikaKolesaRedHT_4:AI_Final_SIP(table:=ADR(kontroller.inputTable)):=(addr:=9, dLL:=0,dHL:=100,dHW:=75,dHA:=80,   histeresis:=0.5, ChangeSIP:=(value:=10));
		//{name:Температура опорного подшипника шестерни редуктора со стороны ЭД т.5 }
		TOpornogoPodshipnikaShesterniReduktoraT_5:AI_Final_SIP(table:=ADR(kontroller.inputTable)):=(addr:=10, dLL:=0,dHL:=100,dHW:=75,dHA:=80,   histeresis:=0.5, ChangeSIP:=(value:=10));
		//{name:Температура опорного подшипника редуктора со стороны Нагнетателя т.6}
		TOpornogoPodshipnikaReduktoraHT_6:AI_Final_SIP(table:=ADR(kontroller.inputTable)):=(addr:=11, dLL:=0,dHL:=100,dHW:=75,dHA:=80,  histeresis:=0.5, ChangeSIP:=(value:=10));
		//{name:Температура опорно-упорного подшипника нагнетателя т.7.1}
		TOpornoYpornogoPodshipnikaNagnetateljaT_7_1:AI_Final_SIP(table:=ADR(kontroller.inputTable)):=(addr:=12, dLL:=0,dHL:=100,dHW:=75,dHA:=80,   histeresis:=0.5, ChangeSIP:=(value:=10));
		//{name:Температура опорно-упорного подшипника нагнетателя т.7.2}
		TOpornoYpornogoPodshipnikaNagnetateljaT_7_2:AI_Final_SIP(table:=ADR(kontroller.inputTable)):=(addr:=13, dLL:=0,dHL:=100,dHW:=75,dHA:=80,  histeresis:=0.5, ChangeSIP:=(value:=10));
		//{name:Температура опорно-упорного подшипника свободного конца нагнетателя т.8.1}
		TOpornoYpornogoPodshipnikaSvobodnogoKoncaNT_8_1:AI_Final_SIP(table:=ADR(kontroller.inputTable)):=(addr:=14, dLL:=0,dHL:=100,dHW:=75,dHA:=80,   histeresis:=0.5, ChangeSIP:=(value:=10));
		//{name:Температура порно-упорного подшипника свободного конца нагнетателя т.8.2}
		TOpornoYpornogoPodshipnikaSvobodnogoKoncaNT_8_2:AI_Final_SIP(table:=ADR(kontroller.inputTable)):=(addr:=15, dLL:=0,dHL:=100,dHW:=75,dHA:=80,   histeresis:=0.5, ChangeSIP:=(value:=10));
		//{name:Температура упорного подшибника рабочих колодок нагнетателя т.9.1}
		TYpornogoPodshipnikaRavKolodokHT_9_1:AI_Final_SIP(table:=ADR(kontroller.inputTable)):=(addr:=16, dLL:=0,dHL:=100,dHW:=75,dHA:=80,   histeresis:=0.5, ChangeSIP:=(value:=10));
		//{name:Температура упорного подшибника рабочих колодок нагнетателя т.9.2}
		TYpornogoPodshipnikaRavKolodokHT_9_2:AI_Final_SIP(table:=ADR(kontroller.inputTable)):=(addr:=17, dLL:=0,dHL:=100,dHW:=75,dHA:=80,   histeresis:=0.5, ChangeSIP:=(value:=10));
		//{name:Температура нерабочих колодок упорного подшипника нагнетателя т.10.1}
		TYpornogoPodshipnikaNerabKolodokHT_10_1:AI_Final_SIP(table:=ADR(kontroller.inputTable)):=(addr:=18, dLL:=0,dHL:=100,dHW:=75,dHA:=80,   histeresis:=0.5, ChangeSIP:=(value:=10));
		//{name:Температура нерабочих колодок упорного подшипника нагнетателя т.10.2}
		TYpornogoPodshipnikaNerabKolodokHT_10_2:AI_Final_SIP(table:=ADR(kontroller.inputTable)):=(addr:=19, dLL:=0,dHL:=100,dHW:=75,dHA:=80,   histeresis:=0.5, ChangeSIP:=(value:=10));
		///////////////////////////////////////////////////////////////////////////////////////////////////////////////
		//{name:Температура холодного воздуха ЭД 1 канал}
		THolodnogoVozduhaEDKanall:AI_Final(table:=ADR(kontroller.inputTable)):=(addr:=20, dLL:=0,dHL:=100, dHW:=60, histeresis:=0.5);
		//{name:Температура холодного воздуха ЭД 2 канал}
		THolodnogoVozduhaEDKanal2:AI_Final(table:=ADR(kontroller.inputTable)):=(addr:=21, dLL:=0,dHL:=100, dHW:=60, histeresis:=0.5);
		
			///////////////////////////////////////////////////////////////////////////////////////////////////////////////
		//{name:Температура горячего воздуха ЭД 1 канал}
		TGorjachegoVozduhaEDKanall:AI_Final(table:=ADR(kontroller.inputTable)):=(addr:=22, dLL:= 0,dHL:=100, dHW:=70, histeresis:=0.5);
		//{name:Температура горячего воздуха ЭД 2 канал}
		TGorjachegoVozduhaEDKanal2:AI_Final(table:=ADR(kontroller.inputTable)):=(addr:=23, dLL:= 0,dHL:=100, dHW:=70, histeresis:=0.5);
		
		//{name:Температура Наружного воздуха}
		TNArujnogoVozduha:AI_Final(table:=ADR(kontroller.inputTable)):=(addr:=24, dLL:=-50,dHL:=100, histeresis:=0.5);
		
		
		
		///////////////////////////////////////////////////////////////////////////////////////////////////////////////
		//{name:Температура газа на входе нагнетателя}
		TgazaNaVhodeH:AI_Final(table:=ADR(kontroller.inputTable)):=(addr:=25, dLL:=-50,dHL:=100,dHW:=80, histeresis:=0.5);
		//{name:Температура газа на выходе нагнетателя}
		TgazaNaVyhodeH:AI_Final_SIP(table:=ADR(kontroller.inputTable)):=(addr:=26, dLL:=-50,dHL:=100,dHW:=80,dHA:=90,   histeresis:=0.5, ChangeSIP:=(value:=10));
		
		///////////////////////////////////////////////////////////////////////////////////////////////////////////////
		//{name:Температура масла до АВОМ}
		TMasladoAVOM:AI_Final(table:=ADR(kontroller.inputTable)):=(addr:=27, dLL:=0,dHL:=150,dHW:=55, histeresis:=0.5);
		//{name:Температура масла после АВОМ}
		TMaslaPosleAVOM:AI_Final_SIP(table:=ADR(kontroller.inputTable)):=(addr:=28, dLL:=0,dHL:=150,dHW:=55,   histeresis:=0.5, ChangeSIP:=(value:=10));
		
		///////////////////////////////////////////////////////////////////////////////////////////////////////////////
		//{name:Температура масла в маслобаке}
		TMaslaMB:AI_Final_SIP(table:=ADR(kontroller.inputTable)):=(addr:=29, dLL:=0,dHL:=150,dLW:=25,   histeresis:=0.5, ChangeSIP:=(value:=10));
		//{name:Температура масла в маслобаке над ТЭН}
		TMaslaMB_TEN:AI_Final_SIP(table:=ADR(kontroller.inputTable)):=(addr:=30, dLL:=0,dHL:=100,dHW:=50,  histeresis:=0.5, ChangeSIP:=(value:=10));
		//{name:Температура в ШУ}
		TEmperatura_v_SHU:AI_Final(table:=ADR(kontroller.inputTable)):=(addr:=32, dLL:=-40,dHL:=100, rassoglasovanie:=2, histeresis:=0.5);
		
		///////////////////////////////////////////////////////////////////////////////////////////////////////////////
		//{name:Давление масла смазки низкое }
		DavlenijaMasloSmNizkoe:AI_Final(table:=ADR(kontroller.inputTable)):=(addr:=33, dLL:=0,dHL:=400,dLW:=50, dLA:=25, rassoglasovanie:=1.5, histeresis:=0.5);
		//{name:Перепад давления масла на масляном фильтре}
		PerepadDavlenieNaMasloFiltre:AI_Final(table:=ADR(kontroller.inputTable)):=(addr:=34, dLL:=0,dHL:=250,dHW:=150, rassoglasovanie:=1.5, histeresis:=0.5);	
		//{name:Давление масла смазки высокое}
		DavlenijaMasloSmVysokoe:AI_Final(table:=ADR(kontroller.inputTable)):=(addr:=35, dLL:=0,dHL:=1000,dLW:=300, dLA:=250, rassoglasovanie:=1.5, histeresis:=0.5);
		//{name:Давление масла смазки после ГНС }
		DavlenijaMaslaPosleGNS:AI_Final(table:=ADR(kontroller.inputTable)):=(addr:=36, dLL:=0,dHL:=1000,dLW:=450, rassoglasovanie:=1.5, histeresis:=0.5);
		//{name:Давление масла после Насоса уплотнения }
		DavlenijaMaslaPosleNU:AI_Final(table:=ADR(kontroller.inputTable)):=(addr:=37, dLL:=0,dHL:=10, dLW:=3, rassoglasovanie:=1.5, histeresis:=0.5);
		///////////////////////////////////////////////////////////////////////////////////////////////////////////////
		
		//{name:Перепад давления газа на Конфузоре}
		PerepadDavlenieNaKonfuzore:AI_Final(table:=ADR(kontroller.inputTable)):=(addr:=40, dLL:=0,dHL:=250, dLW:=15, rassoglasovanie:=1.5, histeresis:=0.5);
		
		/////////////////////////////////////////////////////////////////////////////////////////////////////////////// 
		//{name:Осевой сдвиг нагнетателя +}
		OsSdvigNagnetatelja_Plus:AI_Final(table:=ADR(kontroller.inputTable)):=(addr:=42, dLL:=0,dHL:=1000,dHW:=200, dHA:=300, rassoglasovanie:=1.5, histeresis:=0.5);
		//{name:Осевой сдвиг нагнетателя -}
		OsSdvigNagnetatelja_Minus:AI_Final(table:=ADR(kontroller.inputTable)):=(addr:=43, dLL:=0,dHL:=1000,dHW:=200, dHA:=300, rassoglasovanie:=1.5, histeresis:=0.5); 
		/////////////////////////////////////////////////////////////////////////////////////////////////////////////// 
		//{name:Перепад давления масло-газ }
		PerepadDavlenieMasloGaz:AI_Final(table:=ADR(kontroller.inputTable)):=(addr:=41, dLL:=0,dHL:=1600,dLW:=150, dLA:=100, rassoglasovanie:=1.5);
		///////////////////////////////////////////////////////////////////////////////////////////////////////////////
		//{name:Давление газа на входе нагне-тателя }
		DGazaNaVhodeNagnetatelja:AI_Final(table:=ADR(kontroller.inputTable)):=(addr:=44, dLL:=0,dHL:=10, dLW:=4.895(*, dLA:=4.589*), rassoglasovanie:=1.5, histeresis:=0.5);
		//{name:Давление газа на выходе нагне-тателя }
		DGazaNaVyhodeNagnetatelja:AI_Final(table:=ADR(kontroller.inputTable)):=(addr:=45, dLL:=0, dHL:=10, dHW:=7.55, dHA:=7.653, rassoglasovanie:=1.5, histeresis:=0.5);
		//{name: Давление импульсного газа}
		DavlenieImpulsGaz:AI_Final(table:=ADR(kontroller.inputTable)):=(addr:=46, dLL:=0, dHL:=10, dLW:=5, rassoglasovanie:=1.5, histeresis:=0.5);
		//{name: Уровень масла в маслобаке}
		YrovenMaslaMB:AI_Final(table:=ADR(kontroller.inputTable)):=(addr:=48, dLL:=190,dHL:=885, dLW:=530, rassoglasovanie:=1.5, histeresis:=0.5);
		
		///////////////////////////////////////////////////////////////////////////////////////////////////////////////
		//{name:Контроль ~220В}
		Kontrol_per220V:AI_Final(table:=ADR(kontroller.inputTable)):=(addr:=52, dLL:=0,dHL:=250,dLW:=187,dHW:=242, rassoglasovanie:=1.5, histeresis:=0.5);
		//{name:Контроль =220В}
		Kontrol_post220V:AI_Final(table:=ADR(kontroller.inputTable)):=(addr:=53, dLL:=0,dHL:=250,dLW:=187,dHW:=242, rassoglasovanie:=1.5, histeresis:=0.5);
		
		///////////////////////////////////////////////////////////////////////////////////////////////////////////////
		//{name:Виброскорость опорного подшипника ЭД т.1 }
		VibroSkorostOPED_T1:AI_Final(table:=ADR(kontroller.inputTable)):=(addr:=56, dLL:=0,dHL:=25,dHW:=11, dHA:=18, rassoglasovanie:=1.5, histeresis:=0.5);
		//{name:Виброскорость опорно-упорного подшипника ЭД со стороны редуктора т.2 }
		VibroSkorostOYPED_T2:AI_Final(table:=ADR(kontroller.inputTable)):=(addr:=57, dLL:=0,dHL:=25,dHW:=11, dHA:=18, rassoglasovanie:=1.5, histeresis:=0.5);
		//{name:Виброскорость опорно-упорного подшипника колеса редуктора со стороны ЭД т.3 }
		VibroSkorostOYPKolesaED_T3:AI_Final(table:=ADR(kontroller.inputTable)):=(addr:=58, dLL:=0,dHL:=25,dHW:=11, dHA:=18, rassoglasovanie:=1.5, histeresis:=0.5);
		//{name:Виброскорость опорного подшипника колеса редуктора со стороны нагнетателя т.4 }
		VibroSkorostOPKolesaRH_T4:AI_Final(table:=ADR(kontroller.inputTable)):=(addr:=59, dLL:=0,dHL:=25,dHW:=11, dHA:=18, rassoglasovanie:=1.5, histeresis:=0.5);
		//{name:Виброскорость опорного подшипника шестерни редуктора со стороны ЭД т.5 }
		VibroSkorostOPShesterniRED_T5:AI_Final(table:=ADR(kontroller.inputTable)):=(addr:=60, dLL:=0,dHL:=25,dHW:=11, dHA:=18, rassoglasovanie:=1.5, histeresis:=0.5);
		//{name:Виброскорость опорного подшипника шестерни редуктора со стороны нагнететеля т.6}
		VibroSkorostOPShesterniReduktoraH_T6:AI_Final(table:=ADR(kontroller.inputTable)):=(addr:=61, dLL:=0,dHL:=25,dHW:=11, dHA:=18, rassoglasovanie:=1.5, histeresis:=0.5);
		
		
		
		//{name:Ток статора}
		TokStatora:AI_Final(table:=ADR(kontroller.inputTable)):=(addr:=65, dLL:=0,dHL:=1000,dLW:=300, rassoglasovanie:=1.5, histeresis:=0.5);
		
		
		
		
		///////////////////////////////////////////////////////////////////////////////////////////////////////////////	
	END_STRUCT
END_TYPE

// K2/std12k5/hardwareConfig/DiConfig
TYPE DiConfig:
	STRUCT
		di_0:DiSourceMlp(table:=ADR(kontroller.inputTable)):=(addr:=0);//
		di_1:DiSourceMlp(table:=ADR(kontroller.inputTable)):=(addr:=1);//
		di_2:DiSourceMlp(table:=ADR(kontroller.inputTable)):=(addr:=2);//
		di_3:DiSourceMlp(table:=ADR(kontroller.inputTable)):=(addr:=3);//
		di_4:DiSourceMlp(table:=ADR(kontroller.inputTable)):=(addr:=4);//
		di_5:DiSourceMlp(table:=ADR(kontroller.inputTable)):=(addr:=5);//
		di_6:DiSourceMlp(table:=ADR(kontroller.inputTable)):=(addr:=6);//
		di_7:DiSourceMlp(table:=ADR(kontroller.inputTable)):=(addr:=7);//
		di_8:DiSourceMlp(table:=ADR(kontroller.inputTable)):=(addr:=8);//
		di_9:DiSourceMlp(table:=ADR(kontroller.inputTable)):=(addr:=9);//
		di_10:DiSourceMlp(table:=ADR(kontroller.inputTable)):=(addr:=10);//
		di_11:DiSourceMlp(table:=ADR(kontroller.inputTable)):=(addr:=11);//
		di_12:DiSourceMlp(table:=ADR(kontroller.inputTable)):=(addr:=12);//
		di_13:DiSourceMlp(table:=ADR(kontroller.inputTable)):=(addr:=13);//
		di_14:DiSourceMlp(table:=ADR(kontroller.inputTable)):=(addr:=14);//
		di_15:DiSourceMlp(table:=ADR(kontroller.inputTable)):=(addr:=15);//
		di_16:DiSourceMlp(table:=ADR(kontroller.inputTable)):=(addr:=16);//
		di_17:DiSourceMlp(table:=ADR(kontroller.inputTable)):=(addr:=17);//
		di_18:DiSourceMlp(table:=ADR(kontroller.inputTable)):=(addr:=18);//
		di_19:DiSourceMlp(table:=ADR(kontroller.inputTable)):=(addr:=19);//
		di_20:DiSourceMlp(table:=ADR(kontroller.inputTable)):=(addr:=20);//
		di_21:DiSourceMlp(table:=ADR(kontroller.inputTable)):=(addr:=21);//
	
	END_STRUCT
END_TYPE

// K2/std12k5/algoritms/AlgoritmsConfig
TYPE AlgoritmsConfig:
		{attribute 'symbol' := 'read'}
	STRUCT
		opcComands:OpcCommands(table:=algManager.getTable());
		Auto_Avom_:AutoAVOM (table:=algManager.getTable()):=(T_posle_AVOM:=ai.TMaslaPosleAVOM, A1:=im.v1_Avom, A2:=im.v2_Avom, A3:=im.v3_Avom, A4:=im.v4_Avom);
		autoNu_1:AutoNuAlg_1(table:=algManager.getTable()):=(nu:=Im.nu,di:=im.PerepadDavlenieMasloGaz_Less100, di_CK:=im.PerepadDavlenieMasloGaz_CK);
		autoNu_2:AutoNuAlg_2(table:=algManager.getTable()):=(nu:=Im.nu,di:=im.PerepadDavlenieMasloGaz_Less100, di_CK:=im.PerepadDavlenieMasloGaz_CK);
		autoPns:AutoPnsAlg(table:=algManager.getTable()):=(pns:=Im.pns,Psm_GNS:=ai.DavlenijaMaslaPosleGNS);
		AUto_Ten_:AutoTEn (table:=algManager.getTable()):=(Tmb:=ai.TMaslaMB, TmbTEN:=ai.TMaslaMB_TEN, TEN:=im.TEN_MB, CMN:=im.CMN);
		PNS_ON_MV_:PNS_ON_MV_ON (table:=algManager.getTable()):=(PNS:=im.PNS);
		no:noAlg(table:=algManager.getTable()):=(BlockIm:=FALSE);
		ao:aoAlg(table:=algManager.getTable()):=(BlockIm:=FALSE);
		Opres:Opressovka (table:=algManager.getTable()):=(BlockIm:=FALSE);
		Pms:Prov_Pms (table:=algManager.getTable()):=(BlockIm:=FALSE);
		dPmg:Prov_dPmg (table:=algManager.getTable()):=(BlockIm:=FALSE);
		ppu:ppuAlg(table:=algManager.getTable());
		F1_1:puskFirst_faza1 (table:=algManager.getTable()):=(BlockIm:=FALSE);
		F1_2:puskFirst_faza2 (table:=algManager.getTable()):=(BlockIm:=FALSE);
		F2_Ch:puskSecond_faza_Chastotny (table:=algManager.getTable()):=(BlockIm:=FALSE);
		F2_R:puskSecond_faza_Reactor (table:=algManager.getTable()):=(BlockIm:=FALSE);
		F3:puskThird_faza (table:=algManager.getTable()):=(BlockIm:=FALSE);
		F4:Kran_6_Close (table:=algManager.getTable()):=(BlockIm:=FALSE);
		Kr6_Move: Kran_6_Move (table:=algManager.getTable()):=(BlockIm:=FALSE);
		AutoPNS_Start:PNS_Pusk (table:=algManager.getTable()):=(BlockIm:=FALSE);
		R_AutoAVom:Reset_AutoAVOM (table:=algManager.getTable()):=(BlockIm:=FALSE);
		R_AutoTEN:Reset_AutoTEN (table:=algManager.getTable()):=(BlockIm:=FALSE);
		R_TestIM:Reset_Test_IM (table:=algManager.getTable()):=(BlockIm:=FALSE);
		S_AutoAVOM: Start_AutoAVOM (table:=algManager.getTable()):=(BlockIm:=FALSE);
		S_AutoTEN: Start_AutoTEN (table:=algManager.getTable()):=(BlockIm:=FALSE);
		S_Test_IM: Start_Test_IM (table:=algManager.getTable()):=(BlockIm:=FALSE);
		S_Vibr: Start_ProtectionsVibr(table:=algManager.getTable()):=(BlockIm:=FALSE);
		S_dPmg: Start_Prov_dPmg (table:=algManager.getTable()):=(BlockIm:=FALSE);
		S_I:	Start_Prov_I (table:=algManager.getTable()):=(BlockIm:=FALSE);
		S_K:	Start_Prov_k (table:=algManager.getTable()):=(BlockIm:=FALSE);
		S_Pms:	Start_Prov_Pms (table:=algManager.getTable()):=(BlockIm:=FALSE);
		S_V:	Start_Prov_V (table:=algManager.getTable()):=(BlockIm:=FALSE);
		S_AP:	Start_Pusk_AP (table:=algManager.getTable()):=(BlockIm:=FALSE);
		S_PP:	Start_Pusk_PP (table:=algManager.getTable()):=(BlockIm:=FALSE);
		S_NO:	Start_NO (table:=algManager.getTable()):=(BlockIm:=FALSE);
		S_AO:	Start_AO (table:=algManager.getTable()):=(BlockIm:=FALSE);
		Test_IM: TestIMAlg (table:=algManager.getTable());
		Synch_Rejim_:Synch_Rejims (table:=algManager.getTable());
		Kran4_Samosdvig:Krans_Sdvig_kr4(table:=algManager.getTable()):=(Krans:=im.kran4, block:=ystavki.blockkr4, block_from_alg:=ystavki.Block_kr4_alg);
		Kran1_Samosdvig:Krans_Sdvig_kr4(table:=algManager.getTable()):=(Krans:=im.kran1, block:=ystavki.blockkr1, block_from_alg:=ystavki.Block_kr1_alg); 
		Kran2_Samosdvig:Krans_Sdvig_kr4(table:=algManager.getTable()):=(Krans:=im.kran2, block:=ystavki.blockkr2, block_from_alg:=ystavki.Block_kr2_alg);
		Kran3_Samosdvig:Krans_Sdvig_kr4(table:=algManager.getTable()):=(Krans:=im.kran3, block:=ystavki.blockkr3, block_from_alg:=ystavki.Block_kr3_alg);
		Kran3b_Samosdvig:Krans_Sdvig_kr4(table:=algManager.getTable()):=(Krans:=im.kran3b, block:=ystavki.blockkr3b, block_from_alg:=ystavki.Block_kr3b_alg);
		
		Kran5_Samosdvig:Krans_Sdvig_kr4(table:=algManager.getTable()):=(Krans:=im.kran5, block:=ystavki.blockkr5, block_from_alg:=ystavki.Block_kr5_alg);
		Kran6_Samosdvig:Krans_Sdvig_kr4(table:=algManager.getTable()):=(Krans:=im.kran6, block:=ystavki.blockkr6, block_from_alg:=ystavki.Block_kr6_alg);
		
		Test_P:Test_Protections (table:=algManager.getTable()):=();
		Start_Test_P:Start_Test_Pr (table:=algManager.getTable()):=();
		
	END_STRUCT
END_TYPE

// K2/std12k5/algoritms/ModeGpa
TYPE ModeGpa :
(
	MODE_NOTDEFINED	:= 0, //РЕЖИМ НЕ определен
	MODE_STOP		:= 1, //ГПА остановлен
	MODE_PUSKAP_R	:= 2, //Автоматический пуск Рекакторный
	MODE_PUSKPP_R	:= 3, //Поэтапный пуск Рекакторный
	MODE_PUSKAP_Ch	:= 4, //Автоматический пуск Рекакторный
	MODE_PUSKPP_Ch	:= 5, //Поэтапный пуск Рекакторный
	MODE_WORK_M		:= 6, //Работа в магистраль
	MODE_WORK_K		:= 7, //Работа в кольцо
	MODE_NO			:= 8, //Режим НО
	MODE_AO			:= 9, //Режим АО
	MODE_EO			:= 10, //Режим ЭО
	MODE_TESTIM		:= 11, //Режим тест ИМ
	MODE_PUSKV_R	:= 12, //Режим проверка двигателя в реакторном режиме
	MODE_PUSKV_Ch	:= 13, //Режим проверка двигателя в частотном режиме
	MODE_PUSKK		:= 14, //Режим проверка кранов
	MODE_PROVPMS	:= 15, //Режим проверка давления маслосмазки
	MODE_PROBDPMG	:= 16,	//Режим проверка перепад масло-газ
	MODE_I			:= 17, //режим имитации пуска
	MODE_O			:= 18, //режим опрессовки
	TEST_PROTECTIONS:= 19 //Режим тест защит
) UINT;
END_TYPE

// K2/std12k5/algoritms/ProtectionsConfig
TYPE ProtectionsConfig:
		{attribute 'symbol' := 'read'}
	STRUCT
	(*Температуры т.1 - т.10*) 
		p_TOpornogoPodshipnikaEDT_1:AiProtection (table:=protectManager.getTable())							:=(ai:=ai.TOpornogoPodshipnikaEDT_1	,controlLimit:=statusAi.HA,delay:=(value:=T#3S));
		p_TOpornoYpornogoPodshipnikaEDT_2:AiProtection (table:=protectManager.getTable())					:=(ai:=ai.TOpornoYpornogoPodshipnikaEDT_2 ,controlLimit:=statusAi.HA,delay:=(value:=T#3S));
		p_TOpornoYpornogoPodshipnikaKolesaRedEDT_3:AiProtection (table:=protectManager.getTable())			:=(ai:=ai.TOpornoYpornogoPodshipnikaKolesaRedEDT_3,controlLimit:=statusAi.HA,delay:=(value:=T#3S));
		p_TOpornoYpornogoPodshipnikaKolesaRedHT_4:AiProtection (table:=protectManager.getTable())			:=(ai:=ai.TOpornoYpornogoPodshipnikaKolesaRedHT_4,controlLimit:=statusAi.HA,delay:=(value:=T#3S));
		p_TOpornogoPodshipnikaShesterniReduktoraT_5:AiProtection (table:=protectManager.getTable())			:=(ai:=ai.TOpornogoPodshipnikaShesterniReduktoraT_5	,controlLimit:=statusAi.HA,delay:=(value:=T#3S));
		p_TOpornogoPodshipnikaReduktoraHT_6:AiProtection (table:=protectManager.getTable())					:=(ai:=ai.TOpornogoPodshipnikaReduktoraHT_6,controlLimit:=statusAi.HA,delay:=(value:=T#3S));
		p_TOpornoYpornogoPodshipnikaNagnetateljaT_7:AiProtectionDual (table:=protectManager.getTable())		:=(	ai1:=ai.TOpornoYpornogoPodshipnikaNagnetateljaT_7_1,
																											ai2:=ai.TOpornoYpornogoPodshipnikaNagnetateljaT_7_2	,
																											controlLimit:=statusAi.HA, 
																											control_Normal:=statusAi.Normal, 
																											delay:=(value:=T#3S));
		p_TOpornoYpornogoPodshipnikaSvobodnogoKoncaNT_8:AiProtectionDual (table:=protectManager.getTable())	:=(	ai1:=ai.TOpornoYpornogoPodshipnikaSvobodnogoKoncaNT_8_1,
																											ai2:=ai.TOpornoYpornogoPodshipnikaSvobodnogoKoncaNT_8_2	,
																											controlLimit:=statusAi.HA, 
																											control_Normal:=statusAi.Normal, 
																											delay:=(value:=T#3S));
		p_TYpornogoPodshipnikaRavKolodokHT_9:AiProtectionDual (table:=protectManager.getTable())				:=(	ai1:=ai.TYpornogoPodshipnikaRavKolodokHT_9_1,
																											ai2:=ai.TYpornogoPodshipnikaRavKolodokHT_9_2,
																											controlLimit:=statusAi.HA, 
																											control_Normal:=statusAi.Normal, 
																											delay:=(value:=T#3S));
		p_TYpornogoPodshipnikaNerabKolodokHT_10:AiProtectionDual (table:=protectManager.getTable())				:=(	ai1:=ai.TYpornogoPodshipnikaNerabKolodokHT_10_1,
																											ai2:=ai.TYpornogoPodshipnikaNerabKolodokHT_10_2,
																											controlLimit:=statusAi.HA, 
																											control_Normal:=statusAi.Normal, 
																											delay:=(value:=T#3S));
		p_TgazaNaVyhodeH:AiProtection (table:=protectManager.getTable())									:=(ai:=ai.TgazaNaVyhodeH,controlLimit:=statusAi.HA,delay:=(value:=T#3S));
		
	(*Давления*)
		
		p_OsSdvigNagnetatelja_Plus:AiProtection (table:=protectManager.getTable())							:=(ai:=ai.OsSdvigNagnetatelja_Plus,controlLimit:=statusAi.HA,delay:=(value:=T#3S));
		p_OsSdvigNagnetatelja_Minus:AiProtection (table:=protectManager.getTable())							:=(ai:=ai.OsSdvigNagnetatelja_Minus,controlLimit:=statusAi.HA,delay:=(value:=T#3S));
		p_DGazaNaVhodeNagnetatelja_GPA_STOP:AiProtection (table:=protectManager.getTable())					:=(ai:=ai.DGazaNaVhodeNagnetatelja,controlLimit:=statusAi.normal,ControlValue:=0.3, delay:=(value:=T#3S));
		p_DGazaNaVyhodeNagnetatelja_GPA_STOP:AiProtection (table:=protectManager.getTable())				:=(ai:=ai.DGazaNaVyhodeNagnetatelja,controlLimit:=statusAi.normal,ControlValue:=0.3, delay:=(value:=T#3S));
		//p_DGazaNaVhodeNagnetatelja:AiProtection (table:=protectManager.getTable())							:=(ai:=ai.DGazaNaVhodeNagnetatelja,controlLimit:=statusAi.LA,delay:=(value:=T#3S));
		p_DGazaNaVyhodeNagnetatelja:AiProtection (table:=protectManager.getTable())							:=(ai:=ai.DGazaNaVyhodeNagnetatelja,controlLimit:=statusAi.HA,delay:=(value:=T#3S));
		p_PerepadDavlenieMasloGaz:AiProtection (table:=protectManager.getTable())							:=(ai:=ai.PerepadDavlenieMasloGaz,controlLimit:=statusAi.LA, delay:=(value:=T#20S));
		p_DavlenijaMasloSmNizkoe:AiProtection (table:=protectManager.getTable())							:=(ai:=ai.DavlenijaMasloSmNizkoe,controlLimit:=statusAi.LA, delay:=(value:=T#16S));
		p_DavlenijaMasloSmVysokoe:AiProtection (table:=protectManager.getTable())							:=(ai:=ai.DavlenijaMasloSmVysokoe,controlLimit:=statusAi.LA, delay:=(value:=T#16S));
	
	(*Вибрация*)
		
		p_VibroSkorostOPED_T1:AiProtection (table:=protectManager.getTable())								:=(ai:=ai.VibroSkorostOPED_T1,controlLimit:=statusAi.HA,delay:=(value:=T#3S));
		p_VibroSkorostOYPED_T2:AiProtection (table:=protectManager.getTable())								:=(ai:=ai.VibroSkorostOYPED_T2,controlLimit:=statusAi.HA,delay:=(value:=T#3S));
		p_VibroSkorostOYPKolesaED_T3:AiProtection (table:=protectManager.getTable())						:=(ai:=ai.VibroSkorostOYPKolesaED_T3,controlLimit:=statusAi.HA,delay:=(value:=T#3S));
		p_VibroSkorostOPKolesaRH_T4:AiProtection (table:=protectManager.getTable())							:=(ai:=ai.VibroSkorostOPKolesaRH_T4	,controlLimit:=statusAi.HA,delay:=(value:=T#3S));
		p_VibroSkorostOPShesterniRED_T5:AiProtection (table:=protectManager.getTable())						:=(ai:=ai.VibroSkorostOPShesterniRED_T5	,controlLimit:=statusAi.HA,delay:=(value:=T#3S));
		p_VibroSkorostOPShesterniReduktoraH_T6:AiProtection (table:=protectManager.getTable())				:=(ai:=ai.VibroSkorostOPShesterniReduktoraH_T6,controlLimit:=statusAi.HA,delay:=(value:=T#3S));
	(*Дискретные сигналы *)
		
		p_PerepadDavlenieMasloGaz_Less100:DiProtection (table:=protectManager.getTable())					:=(di:=Im.PerepadDavlenieMasloGaz_Less100,when:=TRUE, delay:=(value:=T#20S));
		p_RegVozbOff:DiProtection (table:=protectManager.getTable())										:=(di:=Im.RegVozbOff, when:=TRUE,delay:=(value:=T#3S));
		p_Fail_Chastotniy_Pusk:DiProtection (table:=protectManager.getTable())								:=(di:=Im.Fail_Chastotniy_Pusk, when:=TRUE,delay:=(value:=T#1S));
		p_OFFAvarSwitch:DiProtection (table:=protectManager.getTable())										:=(di:=Im.OFFAvarSwitch,when:=TRUE,delay:=(value:=T#1S));
		p_AOKC_SHKC:DiProtection (table:=protectManager.getTable())											:=(di:=Im.AOKC_SHKC	,when:=TRUE,delay:=(value:=T#1S));
		p_AO_PRU:DiProtection (table:=protectManager.getTable())											:=(di:=Im.AO_PRU	,when:=TRUE);
		p_AO_fromSHU:DiProtection (table:=protectManager.getTable())										:=(di:=Im.AO_fromSHU	,when:=TRUE);	
					
(*Защиты по ИМ *)																							
		p_mvOff:MvProtection(table:=protectManager.getTable())												:=(sw:=Im.mv,delay:=(value:=T#1S));
		p_kran1:Krans_Protections(table:=protectManager.getTable())											:=(Krans:=Im.kran1, delay:=(value:=T#10S), dP_Konf:=ystavki.dP_Konf_kr1);
		p_kran2:Krans_Protections(table:=protectManager.getTable())											:=(Krans:=Im.kran2, delay:=(value:=T#10S), dP_Konf:=ystavki.dP_Konf_kr1);
		
	END_STRUCT
END_TYPE

// K2/std12k5/modbus/MbsConfig
TYPE MbsConfig:
	STRUCT
		devName:tstModbus(table:=ADR(kontrollers)):=(mbRole:=MbKontrollerRole.MK_SLAVE);

	END_STRUCT
END_TYPE

// Elpk_03_02_COMMON/T_DI03
TYPE T_DI03 :
STRUCT
   {attribute 'displaymode':='hex'}
	In:WORD;// входное (упакованный код из дискр УСО 16 бит)
   {attribute 'displaymode':='hex'}
	A: WORD;// аппаратное
   {attribute 'displaymode':='hex'}
	RR:WORD;// реальное
   {attribute 'displaymode':='hex'}
	R0:WORD;// реальное на предыд такте
//	Vera:REAL;// Veracity - достоверность
	Vera:WORD;// Veracity - достоверность - 25.09.12
	VeraB:BOOL;// Veracity - достоверность - 25.09.12


//	MaskOR:WORD;// маска лог. сложения (In OR mask = A)
// 	MaskOR_flag:BOOL;// флаг необходимости расчета маски лог. сложения
//	
//	MaskAND:WORD;// маска лог. умножения (In AND mask = A)
// 	MaskAND_flag:BOOL;// флаг необходимости расчета маски лог. умножения
//	
//	MaskXOR:WORD;// маска инверсии (In XOR mask = A)
// 	MaskXOR_flag:BOOL;// флаг необходимости расчета маски инверсии

	
	
   {attribute 'displaymode':='hex'}
	Im:WORD;// входное значение, присланное из имтатора (код строки МХ или код DI)
   {attribute 'displaymode':='hex'}
	Imx:WORD;// код перехода в режим имитации для этой переменной (=55AA hex)
			// если код в этом поле = 55AA, то должны использоваться данные из имитатора, а не из УСО
	
	T:DWORD;
	D:DWORD;
	Chg_flag:BOOL;
	
//	EXEC:DI_EXEC1;// программа обработки 
	

END_STRUCT
END_TYPE

// Elpk_03_02_COMMON/T_AI03
TYPE T_AI03 :
STRUCT
	In:WORD;// входное (код АЦП)
	A: REAL;// аппаратное
	RR:REAL;// реальное
	R0:REAL;// реальное на предыд такте
//	Vera:REAL;// Veracity - достоверность
	Vera:WORD;// Veracity - достоверность - 25.09.12
	VeraB:BOOL;// Veracity - достоверность - 25.09.12

	Iv:REAL;// интервал
	Iv_flag:BOOL;// флаг необходимости расчета интервалов по этой переменной
	LL:REAL;// нижняя граница диапазона
	LA:REAL;// нижняя аварийная граница
	LW:REAL;// нижняя предупредительная граница
	HW:REAL;// верхняя предупредительная граница
	HA:REAL;// верхняя аварийная граница
	HL:REAL;// верхняя граница диапазона
// 26 ноя 2013
	dLL:REAL;// дельта для нижней границы диапазона
	dHL:REAL;// дельта для верхней границы диапазона
// 26 ноя 2013
	
	Cmax:REAL;// КОД - верх граница
	Cmin:REAL;// КОД - ниж граница
//	Tmax:REAL;// ФИЗ - верх граница
//	Tmin:REAL;// ФИЗ - ниж граница

	B0:REAL;// сдвиг нуля
	Kx:REAL;// коэффициент (угол наклона)
	Kx_flag:BOOL;// флаг необходимости расчета шкалы по этой переменной
	
(*	Ap:REAL;// аппертура
	Ap_R0:REAL;// предыд значение сигнала
	 Ap_flag:BOOL;// флаг необходимости расчета аппертуры по этой переменной
	  Temp_Ap:REAL;// временный буфер хранения промежуточных результатов Ap
	Pik, Pik_cnt:REAL;
	 Pik_flag:BOOL;// флаг необходимости фильтрации пиков по этой переменной
	  Temp_Pik:REAL;// временный буфер хранения промежуточных результатов Pik
	Ex:REAL;// сглаживание
 	 Ex_flag:BOOL;// флаг необходимости расчета сглаживания по этой переменной
	  Temp_Ex:REAL;// временный буфер хранения промежуточных результатов Ex
////	Gst:REAL;// гистерезис
////	Gst_flag:BOOL;// флаг необходимости расчета гистерезиса по этой переменной   *)
	
	Im:WORD;// входное значение, присланное из имтатора (код АЦП)
   {attribute 'displaymode':='hex'}
	Imx:WORD;// код перехода в режим имитации для этой переменной (=55AA hex)
			// если код в этом поле = 55AA, то должны использоваться данные из имитатора, а не из УСО
		
	T:DWORD;
	D:DWORD;
	Chg_flag:BOOL;
	Rmn_flag:BOOL;// 10.07.13 =T - установлен ремонт AI - на 15 июля 2013 зарезервировано для расширения системы!!!
	
//	EXEC:AI_EXEC1;// программа обработки 
//	EXEC_dLL_dHL:A_dLL_dHL;// программа добавления нижней и верхней дельты    26 ноя 2013

END_STRUCT
END_TYPE

// Elpk_03_02_COMMON/T_DIAGNOSTIC03
TYPE T_DIAGNOSTIC03 :
STRUCT
   {attribute 'displaymode':='hex'}
	CH_MODCONF:WORD;
   {attribute 'displaymode':='hex'}
	CH_ERRNOW:WORD;
   {attribute 'displaymode':='hex'}
	CH_ERRHIST:WORD;
   {attribute 'displaymode':='hex'}
	CH_NDIAG:WORD;
   {attribute 'displaymode':='hex'}
	CH_MDIAG:WORD;
   {attribute 'displaymode':='hex'}
	CH_FIRMVER:WORD;
   {attribute 'displaymode':='hex'}
	CH_FIRMDATE:WORD;
   {attribute 'displaymode':='hex'}
	CH_REZERV7:WORD;	

END_STRUCT
END_TYPE

// Elpk_03_02_COMMON/T_DO03
TYPE T_DO03 :
STRUCT
   {attribute 'displaymode':='hex'}
	In:WORD;// входное (упакованный код из дискр УСО 16 бит)
   {attribute 'displaymode':='hex'}
	A: WORD;// аппаратное
   {attribute 'displaymode':='hex'}
	RR:WORD;// реальное
   {attribute 'displaymode':='hex'}
	R0:WORD;// реальное на предыд такте
//	Vera:REAL;// Veracity - достоверность
	Vera:WORD;// Veracity - достоверность - 25.09.12
	VeraB:BOOL;// Veracity - достоверность - 25.09.12
   {attribute 'displaymode':='hex'}
	Q:WORD;// выход

   {attribute 'displaymode':='hex'}
	Im:WORD;// входное значение, присланное из имтатора (код строки МХ или код DI)
   {attribute 'displaymode':='hex'}
	Imx:WORD;// код перехода в режим имитации для этой переменной (=55AA hex)
			// если код в этом поле = 55AA, то должны использоваться данные из имитатора, а не из УСО
	
	T:DWORD;
	D:DWORD;
	Chg_flag:BOOL;

//	EXEC:DO_EXEC1;// программа обработки 

END_STRUCT
END_TYPE

// K2/std12k5/algoritms/ImConfig
TYPE ImConfig:
	{attribute 'symbol' := 'readwrite'}
	STRUCT
		//u1:singleSignal(table:=ADR(imTable)):=(signal:=di.di_0.bits[0]);
		/////////***КРАНЫ***///////////////////////////////////////////////////////////////
		///////////////////////////////////////////////////////////////////////////////////
		//{name:Кран 1}	
		kran1:Kran(table:=ADR(imTable)):=(
			statOn:=	di.di_20.bits[5].inverse,
			statOff:=	di.di_20.bits[4].inverse,		
			
			cmdOn:=		od.do_0.bits[0],
			cmdOff:=	od.do_0.bits[1],
			
			inSO:=		di.di_16.bits[0].inverse,
			inSZ:=		di.di_16.bits[1].inverse
		);
		///////////////////////////////////////////////////////////////////////////////////
		//{name:Кран 2}	
		kran2:Kran(table:=ADR(imTable)):=(
			statOn:=	di.di_21.bits[0].inverse,
			statOff:=	di.di_20.bits[7].inverse,
			
			cmdOn:=		od.do_0.bits[2],
			cmdOff:=	od.do_0.bits[3], 
			
			inSO:=		di.di_16.bits[2].inverse,
			inSZ:=		di.di_16.bits[3].inverse
			
		);
		///////////////////////////////////////////////////////////////////////////////////
		//{name:Кран 3}	
		kran3:Kran(table:=ADR(imTable)):=(
			statOn:=	di.di_0.bits[5].inverse,
			statOff:=	di.di_0.bits[4].inverse,
			
			cmdOn:=		od.do_0.bits[4],
			cmdOff:=	od.do_0.bits[5],
			
			inSO:=		di.di_16.bits[4].inverse,
			inSZ:=		di.di_16.bits[5].inverse
		);
		///////////////////////////////////////////////////////////////////////////////////
		//{name:Кран 3'}	
		kran3b:Kran(table:=ADR(imTable)):=(
			statOn:=	di.di_0.bits[7].inverse,
			statOff:=	di.di_0.bits[6].inverse,
			
			cmdOn:=		od.do_0.bits[6],
			cmdOff:=	od.do_0.bits[7],
			
			inSO:=		di.di_16.bits[6].inverse,
			inSZ:=		di.di_16.bits[7].inverse
		);	
		///////////////////////////////////////////////////////////////////////////////////
		//{name:Кран 4}	
		kran4:Kr4(table:=ADR(imTable)):=(
			statOn:=	di.di_1.bits[1].inverse,
			statOff:=	di.di_1.bits[0].inverse,
			
			cmdOn:=		od.do_0.bits[8],
			cmdOff:=	od.do_0.bits[9],
			
			inSO:=		di.di_17.bits[0].inverse,
			inSZ:=		di.di_17.bits[1].inverse
		);	
		///////////////////////////////////////////////////////////////////////////////////
		//{name:Кран 5}	
		kran5:Kran(table:=ADR(imTable)):=(
			statOn:=	di.di_1.bits[3].inverse,
			statOff:=	di.di_1.bits[2].inverse,
			
			cmdOn:=		od.do_0.bits[10],
			cmdOff:=	od.do_0.bits[11],
			
			inSO:=		di.di_17.bits[2].inverse,
			inSZ:=		di.di_17.bits[3].inverse
		);	

		///////////////////////////////////////////////////////////////////////////////////
		//{name:Кран 6}	
		kran6:Kran(table:=ADR(imTable)):=(
			statOn:=	di.di_1.bits[5].inverse,
			statOff:=	di.di_1.bits[4].inverse,		
			
			cmdOn:=		od.do_0.bits[12],
			cmdOff:=	od.do_0.bits[13],
			
			inSO:=		di.di_17.bits[4].inverse,
			inSZ:=		di.di_17.bits[5].inverse
		);
		
		
		
		/////////***ИМ***//////////////////////////////////////////////////////////////////
		///////////////////////////////////////////////////////////////////////////////////
		//{name:МВ}	
		mv:SectionSwitch(table:=ADR(imTable)):=(
			statOn:=	di.di_7.bits[0],
			statOff:=	di.di_20.bits[3],
			
			basketRolledIn:= di.di_7.bits[2].inverse,
			basketRolledOut:= di.di_7.bits[2],
			
			cmdOn:=		od.do_4.bits[6],
			cmdOff:=	od.do_4.bits[7]
		);
		///////////////////////////////////////////////////////////////////////////////////
		//{name:В1 АВОМ}	
		v1_Avom:Avom1(table:=ADR(imTable)):=(
			statOn:=	di.di_5.bits[3],
			statOff:=	di.di_5.bits[3]._inversed,
			
			cmdOn:=		od.do_1.bits[8],
			cmdOff:=	od.do_1.bits[9]
		);		
		///////////////////////////////////////////////////////////////////////////////////
		//{name:В2 АВОМ}	
		v2_Avom:Avom2(table:=ADR(imTable)):=(
			statOn:=	di.di_5.bits[4],
			statOff:=	di.di_5.bits[4]._inversed,
			
			cmdOn:=		od.do_1.bits[10],
			cmdOff:=	od.do_1.bits[11]
			
		);	
		///////////////////////////////////////////////////////////////////////////////////
		//{name:В3 АВОМ}	
		v3_Avom:Avom3(table:=ADR(imTable)):=(
			statOn:=	di.di_5.bits[5],
			statOff:=	di.di_5.bits[5]._inversed,
			
			cmdOn:=		od.do_1.bits[12],
			cmdOff:=	od.do_1.bits[13]
		);		
		///////////////////////////////////////////////////////////////////////////////////
		//{name:В4 АВОМ}	
		v4_Avom:Avom4(table:=ADR(imTable)):=(
			statOn:=	di.di_5.bits[6],
			statOff:=	di.di_5.bits[6]._inversed,
			
			cmdOn:=		od.do_1.bits[14],
			cmdOff:=	od.do_1.bits[15]
		);	
		///////////////////////////////////////////////////////////////////////////////////
		//{name:ТЭН МБ}	
		TEN_MB:TEN_MB_(table:=ADR(imTable)):=(	
			statOn:=	di.di_10.bits[0],
			statOff:=	di.di_10.bits[0]._inversed,
			
			cmdOn:=		od.do_2.bits[2],
			cmdOff:=	od.do_2.bits[3] 
		);		
		///////////////////////////////////////////////////////////////////////////////////
		//{name:ТЭН Коллектора}	
		TEN_Kollectira:TEN_Kollectora_(table:=ADR(imTable)):=(	
			statOn:=	di.di_10.bits[1],
			statOff:=	di.di_10.bits[1]._inversed,
			
			cmdOn:=		od.do_2.bits[6],
			cmdOff:=	od.do_2.bits[7]
		);		
		///////////////////////////////////////////////////////////////////////////////////
		//{name:ЦМН}	
		CMN:CMN_(table:=ADR(imTable)):=(	
			statOn:=	di.di_10.bits[3],
			statOff:=	di.di_10.bits[3]._inversed,
			
			cmdOn:=		od.do_2.bits[4],
			cmdOff:=	od.do_2.bits[5]
		);		
		///////////////////////////////////////////////////////////////////////////////////
		//{name:ПНС}	
		PNS:PNS_(table:=ADR(imTable)):=(	
			statOn:=	di.di_5.bits[0],
			statOff:=	di.di_5.bits[0]._inversed,
			
			cmdOn:=		od.do_1.bits[0],
			cmdOff:=	od.do_1.bits[1]
		);		
		///////////////////////////////////////////////////////////////////////////////////
		//{name:НУ}
		nu:NasosNu(table:=ADR(imTable)):=(
			nu1:=(	
				statOn:=	di.di_5.bits[1],
				statOff:=	di.di_5.bits[1]._inversed,
				
				cmdOn:=		od.do_1.bits[4],
				cmdOff:=	od.do_1.bits[5]
			),			

			nu2:=(	
				statOn:=	di.di_5.bits[2],
				statOff:=	di.di_5.bits[2]._inversed,
				
				cmdOn:=		od.do_1.bits[6],
				cmdOff:=	od.do_1.bits[7]
			)
				
		);
		///////////////////////////////////////////////////////////////////////////////////
		//{name:Калорифер АВОмасла}
		KaloriferAVOM:Kalorifer_AVOM_(table:=ADR(imTable)):=(	
			statOn:=	di.di_10.bits[2],
			statOff:=	di.di_10.bits[2]._inversed,
			
			cmdOn:=		od.do_2.bits[0],
			cmdOff:=	od.do_2.bits[1]
		);		

		
		
		
		/////////***Дискреты***//////////////////////////////////////////////////////////////////
		///////////Перепад Давления Масло-газ////////////////////////////////////////////////////////////////////////
		//{name:Перепад давления масло-газ  < 100 кПа}
		PerepadDavlenieMasloGaz_Less100:singleSignal(table:=ADR(imTable)):=(signal:=di.di_20.bits[6]);
		//{name:Обрыв сигнала "Перепад давления масло-газ  > 100 кПа"}
		PerepadDavlenieMasloGaz_NS:Reability(table:=ADR(imTable)):=(di1:=di.di_4.bits[0], when:=FALSE);
		//{name:Наличие ЦК "Перепад давления масло-газ  > 100 кПа"}
		PerepadDavlenieMasloGaz_CK:Reability(table:=ADR(imTable)):=(di1:=di.di_4.bits[0], when:=TRUE);	
		
		///////////Перепад На кране 1////////////////////////////////////////////////////////////////////////	
		//{name:Перепад давления на кране 1 < 100 кПа}
		PerepadDavlenieKran1_Less100:singleSignal(table:=ADR(imTable)):=(signal:=di.di_4.bits[1]);
		//{name:Обрыв сигнала "Перепад давления на кране 1 < 100 кПа"}
		PerepadDavlenieKran1_NS:Reability(table:=ADR(imTable)):=(di1:=di.di_4.bits[1], when:=FALSE);
		//{name:Наличие ЦК "Перепад давления на кране 1 < 100 кПа"}
		PerepadDavlenieKran1_CK:Reability(table:=ADR(imTable)):=(di1:=di.di_4.bits[1],  when:=TRUE);
		
		///////////Отклонение уровня масла в аккумуляторе уплотнения////////////////////////////////////////////////////////////////////////
		//{name:Отклонение уровня масла в аккумуляторе уплотнения} 
		LevelMaslaAkkum:ims(table:=ADR(imTable)):=(di1:=di.di_4.bits[2], di2:=di.di_4.bits[2]);
		//{name:Обрыв сигнала "Отклонение уровня масла в аккумуляторе уплотнения"} 
		LevelMaslaAkkum_NS:Reability(table:=ADR(imTable)):=(di1:=di.di_4.bits[2], when:=FALSE);
		//{name:Наличие ЦК "Отклонение уровня масла в аккумуляторе уплотнения"} 
		LevelMaslaAkkum_CK:Reability(table:=ADR(imTable)):=(di1:=di.di_4.bits[2],  when:=TRUE);
		
		///////////Разрешение загрузки двигателя////////////////////////////////////////////////////////////////////////
		//{name:Разрешение загрузки двигателя}
		LoadDriveisGranted:singleSignal(table:=ADR(imTable)):=(signal:=di.di_6.bits[1]);
		//{name:Обрыв сигнала "Разрешение загрузки двигателя"}
		LoadDriveisGranted_NS:Reability(table:=ADR(imTable)):=(di1:=di.di_6.bits[1], when:=FALSE);
		//{name:Наличие ЦК "Разрешение загрузки двигателя"}
		LoadDriveisGranted_CK:Reability(table:=ADR(imTable)):=(di1:=di.di_6.bits[1], when:=TRUE);
		
		///////////Готовность возбудителя////////////////////////////////////////////////////////////////////////
		//{name:Готовность возбудителя}
		VozbutetelisReady:singleSignal(table:=ADR(imTable)):=(signal:=di.di_6.bits[0]);
		//{name:Обрыв сигнала "Готовность возбудителя"}
		VozbutetelisReady_NS :Reability(table:=ADR(imTable)):=(di1:=di.di_6.bits[0], when:=FALSE);
		//{name:Наличие ЦК "Готовность возбудителя"}
		VozbutetelisReady_CK :Reability(table:=ADR(imTable)):=(di1:=di.di_6.bits[0], when:=TRUE);
		
		///////////Неисправность возбудителя////////////////////////////////////////////////////////////////////////
		//{name:Останов по защитам возбудителя (авария)}
		RegVozbOff:singleSignal(table:=ADR(imTable)):=(signal:=di.di_21.bits[7]);
		//{name:Обрыв сигнала "Останов по защитам возбудителя (авария)"}
		RegVozbOff_NS:Reability(table:=ADR(imTable)):=(di1:=di.di_6.bits[2], when:=FALSE);
		//{name:Наличие ЦК  "Останов по защитам возбудителя (авария)"}
		RegVozbOff_CK:Reability(table:=ADR(imTable)):=(di1:=di.di_6.bits[2], when:=TRUE);
		
		///////////Отключение основного регулятора (неисправность)////////////////////////////////////////////////////////////////////////
		//{name:Отключение основного регулятора (неисправность)}
		MainRegOff:singleSignal(table:=ADR(imTable)):=(signal:=di.di_6.bits[3]);
		//{name:Обрыв сигнала "тключение основного регулятора (неисправность)"}
		MainRegOff_NS:Reability(table:=ADR(imTable)):=(di1:=di.di_6.bits[3], when:=FALSE);
		//{name:Наличие ЦК "тключение основного регулятора (неисправность)"}
		MainRegOff_CK:Reability(table:=ADR(imTable)):=(di1:=di.di_6.bits[3], when:=TRUE);
		
		///////////Неисправность цепей управления АВР питания возбудителя////////////////////////////////////////////////////////////////////////
		//{name:Неисправность цепей управления АВР питания возбудителя}
		AVR_Vozb_Malfanctional:singleSignal(table:=ADR(imTable)):=(signal:=di.di_6.bits[4]);
		//{name:Обрыв сигнала "Неисправность цепей управления АВР питания возбудителя"}
		AVR_Vozb_Malfanctional_NS:Reability(table:=ADR(imTable)):=(di1:=di.di_6.bits[4], when:=FALSE);
		//{name:Наличие ЦК "Неисправность цепей управления АВР питания возбудителя"}
		AVR_Vozb_Malfanctional_CK:Reability(table:=ADR(imTable)):=(di1:=di.di_6.bits[4], when:=TRUE);
		
		///////////Аварийное выключение выключателя////////////////////////////////////////////////////////////////////////
		//{name:Аварийное отключение выключателя}
		OFFAvarSwitch:singleSignal(table:=ADR(imTable)):=(signal:=di.di_8.bits[0]);
		//{name:Обрыв сигнала "Аварийное отключение выключателя"}
		OFFAvarSwitch_NS:Reability(table:=ADR(imTable)):=(di1:=di.di_8.bits[0], when:=FALSE);
		//{name:Наличие ЦК "Аварийное отключение выключателя"}
		OFFAvarSwitch_CK:Reability(table:=ADR(imTable)):=(di1:=di.di_8.bits[0], when:=TRUE);
		
		///////////Асинхронный ход перегрузка////////////////////////////////////////////////////////////////////////
		//{name:Асинхронный ход перегрузка}
		AsynchronnyHod:singleSignal(table:=ADR(imTable)):=(signal:=di.di_8.bits[1]);
		//{name:Обрыв сигнала "Асинхронный ход перегрузка"}
		AsynchronnyHod_NS:Reability(table:=ADR(imTable)):=(di1:=di.di_8.bits[1], when:=FALSE);
		//{name:Наличие ЦК  "Асинхронный ход перегрузка"}
		AsynchronnyHod_CK:Reability(table:=ADR(imTable)):=(di1:=di.di_8.bits[1], when:=TRUE);
		
		///////////Автомат в ячейке ШУ включен////////////////////////////////////////////////////////////////////////
		//{name:Автомат в ячейке ШУ включен}
		Avtomat_SHU_on:singleSignal(table:=ADR(imTable)):=(signal:=di.di_8.bits[2]);
		//{name:Обрыв сигнала "Автомат в ячейке ШУ включен"}
		Avtomat_SHU_on_NS:Reability(table:=ADR(imTable)):=(di1:=di.di_8.bits[2], when:=FALSE);
		//{name:Наличие ЦК  "Автомат в ячейке ШУ включен"}
		Avtomat_SHU_on_CK:Reability(table:=ADR(imTable)):=(di1:=di.di_8.bits[2], when:=TRUE);
		
		///////////Автомат в ШП включен////////////////////////////////////////////////////////////////////////
		//{name:Автомат ШП включен}
		Avtomat_SHP_on:singleSignal(table:=ADR(imTable)):=(signal:=di.di_8.bits[3]);
		//{name:Обрыв сигнала "Автомат ШП включен"}
		Avtomat_SHP_on_NS:Reability(table:=ADR(imTable)):=(di1:=di.di_8.bits[3], when:=FALSE);
		//{name:Наличие ЦК "Автомат ШП включен"}
		Avtomat_SHP_on_CK:Reability(table:=ADR(imTable)):=(di1:=di.di_8.bits[3], when:=TRUE);
		
		///////////Напряжение на секции в норме////////////////////////////////////////////////////////////////////////
		//{name:Напряжение на секции в норме}
		U_Sekcii:singleSignal(table:=ADR(imTable)):=(signal:=di.di_8.bits[4]);
		//{name:Обрыв сигнала "Напряжение на секции в норме"}
		U_Sekcii_NS:Reability(table:=ADR(imTable)):=(di1:=di.di_8.bits[4], when:=FALSE);
		//{name:Наличие ЦК "Напряжение на секции в норме"}
		U_Sekcii_CK:Reability(table:=ADR(imTable)):=(di1:=di.di_8.bits[4], when:=TRUE);
		
		///////////Реакторный пуск////////////////////////////////////////////////////////////////////////
		//{name:Реакторный пуск}
		Reactorni_Pusk:singleSignal(table:=ADR(imTable)):=(signal:=di.di_8.bits[5]);
		//{name:Обрыв сигнала "Напряжение на секции в норме"}
		Reactorni_Pusk_NS:Reability(table:=ADR(imTable)):=(di1:=di.di_8.bits[5], when:=FALSE);
		//{name:Наличие ЦК "Напряжение на секции в норме"}
		Reactorni_Pusk_CK:Reability(table:=ADR(imTable)):=(di1:=di.di_8.bits[5], when:=TRUE);
		
		///////////Частотный пуск////////////////////////////////////////////////////////////////////////
		//{name:Частотный пуск}
		Chastotniy_Pusk:singleSignal(table:=ADR(imTable)):=(signal:=di.di_9.bits[0]);
		//{name:Обрыв сигнала "Частотный пуск"}
		Chastotniy_Pusk_NS:Reability(table:=ADR(imTable)):=(di1:=di.di_9.bits[0], when:=FALSE);
		//{name:Наличие ЦК "Частотный пуск"}
		Chastotniy_Pusk_CK:Reability(table:=ADR(imTable)):=(di1:=di.di_9.bits[0], when:=TRUE);
		
		///////////Неуспешный Частотный пуск////////////////////////////////////////////////////////////////////////
		//{name:Неуспешный Частотный пуск}
		Fail_Chastotniy_Pusk:singleSignal(table:=ADR(imTable)):=(signal:=di.di_9.bits[1]);
		//{name:Обрыв сигнала "Неуспешный Частотный пуск"}
		Fail_Chastotniy_Pusk_NS:Reability(table:=ADR(imTable)):=(di1:=di.di_9.bits[1], when:=FALSE);
		//{name:Наличие ЦК "Неуспешный Частотный пуск"}
		Fail_Chastotniy_Pusk_CK:Reability(table:=ADR(imTable)):=(di1:=di.di_9.bits[1], when:=TRUE);
		
		///////////Режим ручного регулирования////////////////////////////////////////////////////////////////////////
		//{name:Режим ручного регулирования}
		Hand_Reg_rej:singleSignal(table:=ADR(imTable)):=(signal:=di.di_9.bits[2]);
		//{name:Обрыв сигнала "Режим ручного регулирования"}
		Hand_Reg_rej_NS:Reability(table:=ADR(imTable)):=(di1:=di.di_9.bits[2], when:=FALSE);
		//{name:Наличие ЦК "Режим ручного регулирования"}
		Hand_Reg_rej_CK:Reability(table:=ADR(imTable)):=(di1:=di.di_9.bits[2], when:=TRUE);
		
		///////////АО КЦ от ШКС-04М////////////////////////////////////////////////////////////////////////
		//{name:АО КЦ от ШКС-04М}
		AOKC_SHKC:singleSignal(table:=ADR(imTable)):=(signal:=di.di_20.bits[0]);
		//{name:Обрыв сигнала "АО КЦ от ШКС-04М"}
		AOKC_SHKC_NS:Reability(table:=ADR(imTable)):=(di1:=di.di_9.bits[3], when:=FALSE);
		//{name:Наличие ЦК "АО КЦ от ШКС-04М"}
		AOKC_SHKC_CK:Reability(table:=ADR(imTable)):=(di1:=di.di_9.bits[3], when:=TRUE);
		
		///////////НО ГПА от кнопки на ШУ////////////////////////////////////////////////////////////////////////
		//{name:НО ГПА от кнопки на ШУ}
		NO_fromSHU:singleSignal(table:=ADR(imTable)):=(signal:=di.di_21.bits[1]);
		//{name:Обрыв сигнала "НО ГПА от кнопки на ШУ"}
		NO_fromSHU_NS:Reability(table:=ADR(imTable)):=(di1:=di.di_9.bits[4], when:=FALSE);
		//{name:Наличие ЦК  "НО ГПА от кнопки на ШУ"}
		NO_fromSHU_CK:Reability(table:=ADR(imTable)):=(di1:=di.di_9.bits[4], when:=TRUE);
		
		///////////АО ГПА от кнопки на ШУ////////////////////////////////////////////////////////////////////////
		//{name:АО ГПА от кнопки на ШУ}
		AO_fromSHU:singleSignal(table:=ADR(imTable)):=(signal:=di.di_21.bits[2]);
		//{name:Обрыв сигнала "АО ГПА от кнопки на ШУ"}
		AO_fromSHU_NS:Reability(table:=ADR(imTable)):=(di1:=di.di_9.bits[5], when:=FALSE);
		//{name:Наличие ЦК  "АО ГПА от кнопки на ШУ"}
		AO_fromSHU_CK:Reability(table:=ADR(imTable)):=(di1:=di.di_9.bits[5], when:=TRUE);
		
		///////////АО ЭГПА от ПРУ////////////////////////////////////////////////////////////////////////
		//{name:АО ЭГПА от ПРУ}
		AO_PRU:singleSignal(table:=ADR(imTable)):=(signal:=di.di_21.bits[3]);
		//{name:Обрыв сигнала "АО ЭГПА от ПРУ"}
		AO_PRU_NS:Reability(table:=ADR(imTable)):=(di1:=di.di_9.bits[6], when:=FALSE);
		//{name:Наличие ЦК "АО ЭГПА от ПРУ"}
		AO_PRU_CK:Reability(table:=ADR(imTable)):=(di1:=di.di_9.bits[6], when:=TRUE);
		
		///////////НКУ ввод 1 включен////////////////////////////////////////////////////////////////////////
		//{name:НКУ ввод 1 включен}
		NKU_1_On:singleSignal(table:=ADR(imTable)):=(signal:=di.di_10.bits[4]);
		//{name:Обрыв сигнала "НКУ ввод 1 включен"}
		NKU_1_On_NS:Reability(table:=ADR(imTable)):=(di1:=di.di_10.bits[4], when:=FALSE);
		//{name:Наличие ЦК  "НКУ ввод 1 включен"}
		NKU_1_On_CK:Reability(table:=ADR(imTable)):=(di1:=di.di_10.bits[4], when:=TRUE);
		
		///////////НКУ ввод 2 включен////////////////////////////////////////////////////////////////////////
		//{name:НКУ ввод 2 включен}
		NKU_2_On:singleSignal(table:=ADR(imTable)):=(signal:=di.di_10.bits[5]);
		//{name:Обрыв сигнала "НКУ ввод 2 включен"}
		NKU_2_On_NS:Reability(table:=ADR(imTable)):=(di1:=di.di_10.bits[5], when:=FALSE);
		//{name:Наличие ЦК  "НКУ ввод 2 включен"}
		NKU_2_On_CK:Reability(table:=ADR(imTable)):=(di1:=di.di_10.bits[5], when:=TRUE);
		///////////Неисправность цепей контроля ИМ////////////////////////////////////////////////////////////////////////
		MVvkl_Obryv_CK_NS:Reability(table:=ADR(imTable)):=(di1:=di.di_7.bits[0], when:=FALSE);
		MVvykl_Obryv_CK_NS:Reability(table:=ADR(imTable)):=(di1:=di.di_7.bits[1], when:=FALSE);
		MVControl_Work_Obryv_CK_NS:Reability(table:=ADR(imTable)):=(di1:=di.di_7.bits[2], when:=FALSE);
		PNS_vkl_CK_NS:Reability(table:=ADR(imTable)):=(di1:=di.di_5.bits[0], when:=FALSE);
		NU1_vkl_CK_NS:Reability(table:=ADR(imTable)):=(di1:=di.di_5.bits[1], when:=FALSE);
		NU2_vkl_CK_NS:Reability(table:=ADR(imTable)):=(di1:=di.di_5.bits[2], when:=FALSE);
		AVOM1_vkl_CK_NS:Reability(table:=ADR(imTable)):=(di1:=di.di_5.bits[3], when:=FALSE);
		AVOM2_vkl_CK_NS:Reability(table:=ADR(imTable)):=(di1:=di.di_5.bits[4], when:=FALSE);
		AVOM3_vkl_CK_NS:Reability(table:=ADR(imTable)):=(di1:=di.di_5.bits[5], when:=FALSE);
		AVOM4_vkl_CK_NS:Reability(table:=ADR(imTable)):=(di1:=di.di_5.bits[6], when:=FALSE);
		TEN_MB_vkl_CK_NS:Reability(table:=ADR(imTable)):=(di1:=di.di_10.bits[0], when:=FALSE);
		TEN_Kollectora_vkl_CK_NS:Reability(table:=ADR(imTable)):=(di1:=di.di_10.bits[1], when:=FALSE);
		Kalorifer_AVOM_vkl_CK_NS:Reability(table:=ADR(imTable)):=(di1:=di.di_10.bits[2], when:=FALSE);
		CMN_vkl_CK_NS:Reability(table:=ADR(imTable)):=(di1:=di.di_10.bits[3], when:=FALSE);
		///////////Наличие цепей контроля ИМ////////////////////////////////////////////////////////////////////////
		MVvkl_NAlichie_CK:Reability(table:=ADR(imTable)):=(di1:=di.di_7.bits[0], when:=TRUE);
		MVvykl_NAlichie_CK:Reability(table:=ADR(imTable)):=(di1:=di.di_7.bits[1], when:=TRUE);
		MVControl_Work_NAlichie_CK:Reability(table:=ADR(imTable)):=(di1:=di.di_7.bits[2], when:=TRUE);
		PNS_vkl_NAlichie_CK:Reability(table:=ADR(imTable)):=(di1:=di.di_5.bits[0], when:=TRUE);
		NU1_vkl_NAlichie_CK:Reability(table:=ADR(imTable)):=(di1:=di.di_5.bits[1], when:=TRUE);
		NU2_vkl_NAlichie_CK:Reability(table:=ADR(imTable)):=(di1:=di.di_5.bits[2], when:=TRUE);
		AVOM1_vkl_NAlichie_CK:Reability(table:=ADR(imTable)):=(di1:=di.di_5.bits[3], when:=TRUE);
		AVOM2_vkl_NAlichie_CK:Reability(table:=ADR(imTable)):=(di1:=di.di_5.bits[4], when:=TRUE);
		AVOM3_vkl_NAlichie_CK:Reability(table:=ADR(imTable)):=(di1:=di.di_5.bits[5], when:=TRUE);
		AVOM4_vkl_NAlichie_CK:Reability(table:=ADR(imTable)):=(di1:=di.di_5.bits[6], when:=TRUE);
		TEN_MB_vkl_NAlichie_CK:Reability(table:=ADR(imTable)):=(di1:=di.di_10.bits[0], when:=TRUE);
		TEN_Kollectora_vkl_NAlichie_CK:Reability(table:=ADR(imTable)):=(di1:=di.di_10.bits[1], when:=TRUE);
		Kalorifer_AVOM_vkl_NAlichie_CK:Reability(table:=ADR(imTable)):=(di1:=di.di_10.bits[2], when:=TRUE);
		CMN_vkl_NAlichie_CK:Reability(table:=ADR(imTable)):=(di1:=di.di_10.bits[3], when:=TRUE);
		///////////Наличие питания////////////////////////////////////////////////////////////////////////
		//{name:Наличие БП1}
		NalichieBP1:singleSignal(table:=ADR(imTable)):=(signal:=di.di_11.bits[0]);
		//{name:Наличие БП2}
		NalichieBP2:singleSignal(table:=ADR(imTable)):=(signal:=di.di_11.bits[1]);
		//{name:Наличие БП3}
		NalichieBP3:singleSignal(table:=ADR(imTable)):=(signal:=di.di_11.bits[2]);
		//{name:Наличие БП4}
		NalichieBP4:singleSignal(table:=ADR(imTable)):=(signal:=di.di_11.bits[3]);
		//{name:Наличие БП5}
		NalichieBP5:singleSignal(table:=ADR(imTable)):=(signal:=di.di_11.bits[4]);
		//{name:Наличие БП6}
		NalichieBP6:singleSignal(table:=ADR(imTable)):=(signal:=di.di_11.bits[5]);
		//{name:Наличие БП7 и БП8}
		NalichieBP7_BP8:singleSignal(table:=ADR(imTable)):=(signal:=di.di_11.bits[6]);
		//{name:Наличие БП9 и БП10}
		NalichieBP9_BP10:singleSignal(table:=ADR(imTable)):=(signal:=di.di_11.bits[7]);
		//{name:Наличие Цепи управления МВ}
		Nalichie_CU_MV:singleSignal(table:=ADR(imTable)):=(signal:=di.di_12.bits[0]);
		//{name:Наличие напряжения  =220 в БРЭО}
		Nalichie220BEAO:singleSignal(table:=ADR(imTable)):=(signal:=di.di_12.bits[1]);
		//{name:Наличие напряжения на входе в ШУ ~220}
		NalichiePer220naVhode:singleSignal(table:=ADR(imTable)):=(signal:=di.di_12.bits[2]);
		//{name:Наличие напряжения на входе в ШУ =220}
		NalichiePost220naVhode:singleSignal(table:=ADR(imTable)):=(signal:=di.di_12.bits[3]);
		//{name:Наличие БП11}
		NalichieBP11:singleSignal(table:=ADR(imTable)):=(signal:=di.di_12.bits[4]);
		//{name:Наличие БП12}
		NalichieBP12:singleSignal(table:=ADR(imTable)):=(signal:=di.di_12.bits[5]);
		
		///////////Отсутствие питания////////////////////////////////////////////////////////////////////////
		//{name:Нет БП1}
		NalichieBP1_NS:singleSignal(table:=ADR(imTable)):=(signal:=di.di_11.bits[0].inverse);
		//{name:Нет БП2}
		NalichieBP2_NS:singleSignal(table:=ADR(imTable)):=(signal:=di.di_11.bits[1].inverse);
		//{name:Нет БП3}
		NalichieBP3_NS:singleSignal(table:=ADR(imTable)):=(signal:=di.di_11.bits[2].inverse);
		//{name:Нет БП4}
		NalichieBP4_NS:singleSignal(table:=ADR(imTable)):=(signal:=di.di_11.bits[3].inverse);
		//{name:Нет БП5}
		NalichieBP5_NS:singleSignal(table:=ADR(imTable)):=(signal:=di.di_11.bits[4].inverse);
		//{name:Нет БП6}
		NalichieBP6_NS:singleSignal(table:=ADR(imTable)):=(signal:=di.di_11.bits[5].inverse);
		//{name:Нет БП7 и БП8}
		NalichieBP7_BP8_NS:singleSignal(table:=ADR(imTable)):=(signal:=di.di_11.bits[6].inverse);
		//{name:Нет БП9 и БП10}
		NalichieBP9_BP10_NS:singleSignal(table:=ADR(imTable)):=(signal:=di.di_11.bits[7].inverse);
		//{name:Нет Цепи управления МВ}
		Nalichie_CU_MV_NS:singleSignal(table:=ADR(imTable)):=(signal:=di.di_12.bits[0].inverse);
		//{name:Нет напряжения  =220 в БРЭО}
		Nalichie220BEAO_NS:singleSignal(table:=ADR(imTable)):=(signal:=di.di_12.bits[1].inverse);
		//{name:Нет напряжения на входе в ШУ ~220}
		NalichiePer220naVhode_NS:singleSignal(table:=ADR(imTable)):=(signal:=di.di_12.bits[2].inverse);
		//{name:Нет напряжения на входе в ШУ =220}
		NalichiePost220naVhode_NS:singleSignal(table:=ADR(imTable)):=(signal:=di.di_12.bits[3].inverse);
		//{name:Нет БП11}
		NalichieBP11_NS:singleSignal(table:=ADR(imTable)):=(signal:=di.di_12.bits[4].inverse);
		//{name:Нет БП12}
		NalichieBP12_NS:singleSignal(table:=ADR(imTable)):=(signal:=di.di_12.bits[5].inverse);
		
		///////////Двери////////////////////////////////////////////////////////////////////////
		//{name:Дверь ШУ открыта Передняя}
		Door_SHU_Front_Open:singleSignal(table:=ADR(imTable)):=(signal:=di.di_13.bits[0]);
		//{name:Дверь ШУ открыта Задняя}
		Door_SHU_Back_Open:singleSignal(table:=ADR(imTable)):=(signal:=di.di_13.bits[1]);
		//{name:БЭАО сработал}
		
		BEAO_Work:singleSignal(table:=ADR(imTable)):=(signal:=di.di_18.bits[1]);
		//{name:Сброс БЭАО}
		//BEAO_Reset:singleSignal(table:=ADR(imTable)):=(signal:=di.di_18.bits[1]);
		///////////ЩАВР////////////////////////////////////////////////////////////////////////
		//{name:ЩАВР ввод 1 включен}
		SHAVR_1_On:singleSignal(table:=ADR(imTable)):=(signal:=di.di_13.bits[6]);
		//{name:ЩАВР ввод 2 включен}
		SHAVR_2_On:singleSignal(table:=ADR(imTable)):=(signal:=di.di_13.bits[7]);
		
		///////////Кнопки Экстренного останова////////////////////////////////////////////////////////////////////////
		//{name:ЭО ГПА от кнопки на ШУ}
		EO_fromSHU:singleSignal(table:=ADR(imTable)):=(signal:=di.di_14.bits[0]);
		//{name:ЭО ЭГПА от ПРУ}
		EO_PRU:singleSignal(table:=ADR(imTable)):=(signal:=di.di_14.bits[1]);
		
		///////////Напряжение на ИМ////////////////////////////////////////////////////////////////////////
		//{name:Наличие напряжения в ЦУ ПНС}
		NalichieU_PNS:singleSignal(table:=ADR(imTable)):=(signal:=di.di_14.bits[2]);
		//{name:Наличие напряжения в ЦУ НУ1}
		NalichieU_NU1:singleSignal(table:=ADR(imTable)):=(signal:=di.di_14.bits[3]);
		//{name:Наличие напряжения в ЦУ НУ2}
		NalichieU_NU2:singleSignal(table:=ADR(imTable)):=(signal:=di.di_14.bits[4]);
		//{name:Наличие напряжения в ЦУ ЦМН}
		NalichieU_CMN:singleSignal(table:=ADR(imTable)):=(signal:=di.di_14.bits[5]);
		
		///////////Нет Напряжения на ИМ////////////////////////////////////////////////////////////////////////
		//{name:Нет напряжения в ЦУ ПНС}
		NET_U_PNS:singleSignal(table:=ADR(imTable)):=(signal:=di.di_10.bits[10].inverse);
		//{name:Нет напряжения в ЦУ НУ1}
		NET_U_NU1:singleSignal(table:=ADR(imTable)):=(signal:=di.di_10.bits[11].inverse);
		//{name:Нет напряжения в ЦУ НУ2}
		NET_U_NU2:singleSignal(table:=ADR(imTable)):=(signal:=di.di_10.bits[12].inverse);
		//{name:Нет напряжения в ЦУ ЦМН}
		NET_U_CMN:singleSignal(table:=ADR(imTable)):=(signal:=di.di_10.bits[13].inverse);
		
		///////////ИМ в Автомате////////////////////////////////////////////////////////////////////////
		//{name:АВОМ1 в автоматическом режиме}
		AVOM1_Automat:singleSignal(table:=ADR(imTable)):=(signal:=di.di_2.bits[0]);
		//{name:АВОМ2 в автоматическом режиме}
		AVOM2_Automat:singleSignal(table:=ADR(imTable)):=(signal:=di.di_2.bits[1]);
		//{name:АВОМ3 в автоматическом режиме}
		AVOM3_Automat:singleSignal(table:=ADR(imTable)):=(signal:=di.di_2.bits[2]);
		//{name:АВОМ4 в автоматическом режиме}
		AVOM4_Automat:singleSignal(table:=ADR(imTable)):=(signal:=di.di_2.bits[3]);
		
		//{name:ПНС в автоматическом режиме}
		PNS_Automat:singleSignal(table:=ADR(imTable)):=(signal:=di.di_2.bits[4]);
		
		//{name:НУ1 в автоматическом режиме}
		NU1_Automat:singleSignal(table:=ADR(imTable)):=(signal:=di.di_2.bits[5]);
		//{name:НУ2 в автоматическом режиме}
		NU2_Automat:singleSignal(table:=ADR(imTable)):=(signal:=di.di_2.bits[6]);
		
		//{name:ТЭН МБ в автоматическом режиме}
		TEN_MB_Automat:singleSignal(table:=ADR(imTable)):=(signal:=di.di_2.bits[7]);
		//{name:ТЭН Коллектора в автоматическом режиме}
		TEN_Kollectora_Automat:singleSignal(table:=ADR(imTable)):=(signal:=di.di_3.bits[0]);
		
		//{name:Калорифер АВОМ в автоматическом режиме}
		KalAVOM_Automat:singleSignal(table:=ADR(imTable)):=(signal:=di.di_3.bits[1]);
		//{name:ЦМН в автоматическом режиме}
		CMN_Automat:singleSignal(table:=ADR(imTable)):=(signal:=di.di_3.bits[2]);
		//{name:СИнхронизация режима К1}
		Synch_rej_K1:singleSignal(table:=ADR(imTable)):=(signal:=di.di_3.bits[5]);
		Synch_rej_K1_Meandr:singleOutput(table:=ADR(imTable)):=(signal:=od.do_3.bits[13]);
		///////////Поток масла после АВОМ////////////////////////////////////////////////////////////////////////
		//{name:Поток масла после АВОМ > 85 л/мин}
		Flow_Ms_PosleAVOM:singleSignal(table:=ADR(imTable)):=(signal:=di.di_18.bits[0].inverse);
		
		/////////***ДИСКРЕТЫ OUTPUT***//////////////////////////////////////////////////////////////////
		///////////////////////////////////////////////////////////////////////////////////
		
	//	Stop_MV_NO:SingleOutput(table:=ADR(imTable)):=(signal:=od.do_4.bits[2], wait_time:=T#4S);
	
		//{name:Работа ЭГПА}
		Work_EGPA:SingleOutput(table:=ADR(imTable)):=(signal:=od.do_4.bits[2]);
		//{name:Неисправность ЭГПА}
		Neispr_EGPA:SingleOutput(table:=ADR(imTable)):=(signal:=od.do_4.bits[0]);
		//{name:Авария ЭГПА}
		Avary_EGPA:SingleOutput(table:=ADR(imTable)):=(signal:=od.do_4.bits[1]);
		//{name:Наличие напряжения лампа на двери}
		U_Lamp_SHU:SingleOutput(table:=ADR(imTable)):=(signal:=od.do_4.bits[3]);
			//{name:Посветка кнопки при АО}
		AO_Knopka_ind:SingleOutput(table:=ADR(imTable)):=(signal:=od.do_4.bits[4]);
		//{name:Пуск в ШУП}
		Pusk_SHUP:SingleOutput(table:=ADR(imTable)):=(signal:=od.do_4.bits[8], wait_time:=T#4S);
		//{name:Останов в ШУП}
		Stop_SHUP:SingleOutput(table:=ADR(imTable)):=(signal:=od.do_4.bits[9], wait_time:=T#4S);
		//{name:Фонарь НО}
		NO_Fonar:SingleOutput(table:=ADR(imTable)):=(signal:=od.do_3.bits[10]);
		//{name:Фонарь ПС}
		PC_Fonar:SingleOutput(table:=ADR(imTable)):=(signal:=od.do_3.bits[9]);
		//{name:Фонарь АС}
		AC_Fonar:SingleOutput(table:=ADR(imTable)):=(signal:=od.do_3.bits[8]);
		//{name:смазка крана 1}
		Kr1_Smazka:SingleOutput(table:=ADR(imTable)):=(signal:=od.do_0.bits[14], wait_time:=T#15S);
		//{name:смазка крана 2}
		Kr2_Smazka:SingleOutput(table:=ADR(imTable)):=(signal:=od.do_0.bits[15], wait_time:=T#15S);
		//{name:Кран 4 открыть из 3 этапа пуска}
		Kr_4_Open_From_Alg:SingleOutput(table:=ADR(imTable)):=(signal:=od.do_0.bits[8]);
		/////////***ДИСКРЕТЫ Неисправности***//////////////////////////////////////////////////////////////////
	
		
		
		/////////***НАличие Цепей контроля***//////////////////////////////////////////////////////////////////
		///////////////////////////////////////////////////////////////////////////////////
		
		
	END_STRUCT
END_TYPE

// lowLevel_ecl/algoritms/phases/DualStateImAction
TYPE DualStateImAction :
(
	on,
	off
);
END_TYPE

// lowLevel_ecl/algoritms/phases/PhaseAlgoritmAction
TYPE PhaseAlgoritmAction :
(
	run,
	reset
);
END_TYPE

